Yaskawa INFORM job: X2_38-47,64(2)(90,0)_HARDOX.JBI

/JOB
//NAME X2_38-47,64(2)(90,0)_HARDOX
//POS
///NPOS 517,517,517,31,0,0
///TOOL 0
///POSTYPE PULSE
///PULSE
C00000=-10776,-116726,-133110,1428,79202,268
C00001=-117551,-99167,-129064,14869,107235,27560
C00002=-118060,-97833,-124544,14759,105287,27149
C00003=-118255,-97731,-122391,14687,104086,26936
C00004=-118255,-99005,-121658,14606,103015,26804
C00005=-118252,-98719,-121832,14623,103261,26835
C00006=-118753,-92238,-119382,14829,105109,26899
C00007=-118252,-98719,-121832,14623,103261,26835
C00008=-117548,-101379,-128390,14732,105732,27372
C00009=-119930,-99721,-129265,15188,107465,26816
C00010=-120369,-98285,-124713,15062,105542,26424
C00011=-120537,-98252,-122491,14975,104264,26206
C00012=-120537,-99415,-121812,14899,103281,26083
C00013=-120552,-99088,-121997,14922,103557,26112
C00014=-120983,-92542,-119530,15124,105413,26206
C00015=-120552,-99088,-121997,14922,103557,26112
C00016=-119945,-101871,-128593,15052,105999,26622
C00017=-126449,-117484,-130445,19479,74849,30062
C00018=-126433,-122162,-123583,20167,68593,29001
C00019=-126700,-111661,-117040,20113,69946,29141
C00020=-126798,-108107,-114012,20160,69935,29102
C00021=-126799,-108400,-113008,20254,69212,28975
C00022=-126718,-108336,-113627,20168,69582,29070
C00023=-124486,-105728,-112699,19107,69790,29924
C00024=-126718,-108336,-113627,20168,69582,29070
C00025=-121607,-132044,-121280,18982,61321,29585
C00026=-106120,-105771,-112642,10491,66484,36125
C00027=-107709,-101450,-111061,11179,67916,35692
C00028=-106120,-105771,-112642,10491,66484,36125
C00029=-113778,-131562,-126460,14735,63009,32904
C00030=-125989,-135705,-128836,15868,81833,-19678
C00031=-122637,-125595,-122855,15098,82666,-18409
C00032=-121382,-121958,-120533,14807,82865,-17952
C00033=-121382,-122071,-118910,14836,81841,-18076
C00034=-121382,-121958,-120533,14807,82865,-17952
C00035=-106979,-143901,-125029,2861,68009,-11090
C00036=-108002,-136905,-123073,3147,70435,-11396
C00037=-106979,-143901,-125029,2861,68009,-11090
C00038=-130918,-93362,-108301,23503,98063,-21430
C00039=-128613,-93045,-108174,23197,97523,-20724
C00040=-130918,-93362,-108301,23503,98063,-21430
C00041=-136165,-97259,-113946,24281,100844,-22722
C00042=-136175,-89641,-119549,25205,107565,-21267
C00043=-114744,-130738,-127344,-18726,86415,24127
C00044=-118651,-123075,-122041,-18017,86194,22796
C00045=-120132,-120263,-119410,-17742,85711,22351
C00046=-120132,-120365,-118339,-17753,85031,22450
C00047=-120131,-120316,-118616,-17749,85218,22423
C00048=-120610,-114014,-116540,-17635,86988,22001
C00049=-120131,-120316,-118616,-17749,85218,22423
C00050=-120535,-116966,-117470,-17658,86102,22155
C00051=-123144,-118008,-117813,-17156,85246,21372
C00052=-120535,-116966,-117470,-17658,86102,22155
C00053=-115268,-126863,-124750,-18631,86672,23904
C00054=-115290,-123417,-132013,-18678,92595,22992
C00055=-123593,-125758,-130163,6995,115060,-67946
C00056=-111289,-112434,-124190,9231,117016,-63234
C00057=-105837,-112853,-120878,9823,114178,-61462
C00058=-105837,-113368,-119803,9744,113264,-61541
C00059=-105837,-112984,-120626,9804,113958,-61481
C00060=-104314,-115180,-121361,9954,113110,-60999
C00061=-105837,-112984,-120626,9804,113958,-61481
C00062=-140180,-156270,-135194,3647,103600,-74458
C00063=-143876,-158808,-133483,2421,103143,-75779
C00064=-143876,-157752,-132173,2418,102880,-75785
C00065=-143876,-158999,-133717,2421,103190,-75779
C00066=-142833,-166242,-135523,2599,100548,-75469
C00067=-143876,-158999,-133717,2421,103190,-75779
C00068=-138517,-137739,-134524,3768,114393,-73549
C00069=-143641,-117492,-131018,10110,103710,-40081
C00070=-127017,-112123,-129453,9078,98380,-24722
C00071=-128303,-122732,-125182,9622,82824,-11347
C00072=-126354,-112603,-118881,9097,83916,-10616
C00073=-125631,-108986,-116438,8904,84188,-10357
C00074=-125631,-109537,-114964,8919,83013,-10441
C00075=-125631,-108986,-116438,8904,84188,-10357
C00076=-110037,-120252,-118594,-5441,76700,-4050
C00077=-111650,-115152,-116920,-4919,78183,-4659
C00078=-110037,-120252,-118594,-5441,76700,-4050
C00079=-125797,-107165,-114352,8951,83863,-10435
C00080=-123589,-104463,-113383,8361,84418,-9668
C00081=-125797,-107165,-114352,8951,83863,-10435
C00082=-128447,-120300,-122969,9661,82730,-11402
C00083=-128462,-115265,-129707,9620,89375,-10895
C00084=-116938,-126430,-125851,-12631,81878,14685
C00085=-119474,-116309,-119688,-11957,82879,13726
C00086=-120416,-112800,-116898,-11714,82830,13413
C00087=-120416,-113088,-115771,-11732,82005,13491
C00088=-121130,-109897,-115487,-11517,83341,13125
C00089=-121652,-107697,-114715,-11371,83913,12898
C00090=-120385,-110630,-116263,-11708,83544,13356
C00091=-116898,-126708,-125088,-12658,81285,14759
C00092=-116961,-121523,-133241,-12544,88781,13978
C00093=-110477,-156196,-127656,-40514,54336,55405
C00094=-116757,-147091,-123275,-37008,53079,52657
C00095=-119129,-143495,-121504,-35581,52690,51595
C00096=-122199,-143523,-121511,-34086,51426,50520
C00097=-119129,-143495,-121504,-35581,52690,51595
C00098=-121389,-143526,-121523,-34489,51757,50806
C00099=-121378,-138155,-118828,-34021,52680,50458
C00100=-121389,-143526,-121523,-34489,51757,50806
C00101=-121337,-120057,-120260,-30579,61379,47564
C00102=-120272,-114318,-116759,-30898,62447,47698
C00103=-120254,-119054,-117181,-31500,60580,48280
C00104=-120272,-114318,-116759,-30898,62447,47698
C00105=-110477,-159292,-131347,-40206,54861,55162
C00106=-115322,-144881,-127675,-10917,26238,44128
C00107=-131784,-127965,-127002,28991,89678,26741
C00108=-120831,-123140,-121731,27130,85392,29797
C00109=-120549,-120601,-118843,27089,84879,29783
C00110=-120549,-120670,-117777,27109,84260,29640
C00111=-120517,-120686,-117908,27101,84315,29665
C00112=-120983,-114470,-115866,27142,86197,29928
C00113=-120517,-120686,-117908,27101,84315,29665
C00114=-121539,-130455,-126219,27290,84728,29379
C00115=-123491,-138727,-133578,17593,86073,29901
C00116=-123873,-130565,-127363,17655,86508,29830
C00117=-124019,-127789,-124130,17687,86001,29706
C00118=-124019,-127817,-123341,17694,85524,29637
C00119=-124041,-127842,-123499,17696,85609,29642
C00120=-124402,-120732,-121277,17740,87868,29843
C00121=-124041,-127842,-123499,17696,85609,29642
C00122=-123895,-130695,-125894,17671,85585,29689
C00123=-123514,-138829,-132098,17610,85158,29761
C00124=-131669,-108309,-130646,31875,113573,61343
C00125=-139138,-132176,-121475,37127,109735,76690
C00126=-136347,-141301,-121131,36509,104575,76083
C00127=-135137,-144527,-120818,36387,102556,75910
C00128=-135139,-143303,-118803,36292,102059,75739
C00129=-135137,-144527,-120818,36387,102556,75910
C00130=-123222,-117207,-112602,33876,112841,80142
C00131=-123302,-123100,-114500,33386,111310,79603
C00132=-123222,-117207,-112602,33876,112841,80142
C00133=-149473,-167599,-122340,40123,93659,70303
C00134=-145955,-169881,-122827,40768,91382,70949
C00135=-149473,-167599,-122340,40123,93659,70303
C00136=-154660,-158984,-124630,39692,100555,70658
C00137=-145602,-129354,-130944,11561,117970,66438
C00138=-141571,-135796,-129141,-17923,112920,58745
C00139=-145358,-145317,-128855,-18021,107261,58200
C00140=-146973,-148537,-128532,-18134,105137,57926
C00141=-146977,-147425,-126561,-18072,104525,58019
C00142=-146951,-147398,-126788,-18082,104677,58005
C00143=-148016,-155121,-128806,-18044,101844,58047
C00144=-146951,-147398,-126788,-18082,104677,58005
C00145=-147811,-154474,-129578,-18071,102659,57998
C00146=-150760,-151393,-128781,-18698,103033,56852
C00147=-147811,-154474,-129578,-18071,102659,57998
C00148=-142197,-142429,-130522,-17697,110344,58914
C00149=-120703,-123129,-132845,19094,121060,67264
C00150=-120658,-146832,-128060,18624,118943,66884
C00151=-120634,-158899,-128202,17585,113113,65913
C00152=-120623,-163194,-128036,17271,110903,65572
C00153=-120623,-161024,-125795,17237,110651,65534
C00154=-120562,-161261,-126266,17282,110799,65580
C00155=-120543,-169070,-128088,16945,108025,65171
C00156=-120562,-161261,-126266,17282,110799,65580
C00157=-120603,-145779,-126506,18564,118536,66834
C00158=-125859,-133715,-124767,32608,106843,81797
C00159=-122845,-142953,-124347,32149,101432,81430
C00160=-121547,-146160,-123992,32074,99345,81353
C00161=-121546,-144979,-121994,32008,98813,81200
C00162=-109812,-115651,-114700,28773,111647,86169
C00163=-109420,-121743,-116686,28433,109829,85843
C00164=-109812,-115651,-114700,28773,111647,86169
C00165=-136113,-171916,-125823,37236,88758,74782
C00166=-132431,-173177,-126093,37775,86796,75630
C00167=-136113,-171916,-125823,37236,88758,74782
C00168=-141699,-164023,-128432,36630,95711,74814
C00169=-125872,-133752,-131219,33440,110189,40846
C00170=-133109,-126295,-132836,15576,121717,-49477
C00171=-134095,-144484,-127159,11413,120192,-39245
C00172=-134095,-142728,-123587,11251,118920,-39381
C00173=-134108,-141028,-121891,11256,119008,-39376
C00174=-115660,-122947,-115610,-13186,126131,-57848
C00175=-119844,-134491,-118750,-17115,121000,-60623
C00176=-133528,-137451,-116046,-34139,108998,-80448
C00177=-134077,-138654,-116284,-35996,107959,-82962
C00178=-134074,-140235,-119255,-36225,108790,-83252
C00179=-128746,-104991,-133081,-28169,117444,-49732
C00180=-123335,-90933,-122081,-14660,102496,-9308
C00181=-120623,-92535,-112214,-7385,88125,11837
C00182=-120622,-94347,-109953,-7392,85821,11972
C00183=-121706,-96320,-109727,-7087,84579,11689
C00184=-119347,-92925,-108176,-7759,85570,12397
C00185=-120623,-94767,-108750,-7400,84873,12029
C00186=-120184,-98406,-104184,11463,70199,-7234
C00187=-120621,-97250,-102226,16251,67423,-11647
C00188=-120622,-96877,-104163,16104,68755,-11460
C00189=-120643,-108357,-118989,16415,66098,-11840
C00190=-67024,-106779,-124945,-13769,92672,20129
C00191=-67015,-109280,-122780,-13735,90127,20415
C00192=-68524,-114997,-123393,-13374,87393,20218
C00193=-67240,-109374,-121326,-13663,89172,20449
C00194=-67101,-109000,-122679,-13716,90193,20379
C00195=-67110,-106486,-124839,-13750,92741,20094
C00196=-120616,-103713,-129855,-8435,78518,79847
C00197=-120615,-108904,-127553,-8566,74477,80127
C00198=-120827,-110646,-126375,-8530,72852,80171
C00199=-120813,-110572,-126430,-8535,72927,80169
C00200=-120709,-110247,-126307,-8582,73030,80199
C00201=-120779,-110557,-126444,-8550,72945,80181
C00202=-120615,-108909,-127550,-8566,74473,80128
C00203=-118661,-125998,-116417,-35444,53464,49551
C00204=-120918,-122974,-114552,-34038,52889,48644
C00205=-120869,-128815,-114683,-35350,50480,49611
C00206=-120575,-146473,-114035,-40240,44023,53993
C00207=-120599,-119966,-113452,-30276,65744,57931
C00208=-118319,-121507,-115012,-31110,66714,58605
C00209=-113281,-124998,-118777,-32819,69049,60013
C00210=-113467,-117261,-128448,-33027,70743,59318
C00211=-117537,-116112,-134646,-12805,84442,25722
C00212=-120610,-126431,-125414,1040,80197,3464
C00213=-120610,-126707,-122448,1046,78230,3447
C00214=-122238,-127010,-121321,1494,77406,2886
C00215=-120610,-126687,-121221,1049,77486,3441
C00216=-120610,-126294,-121087,1045,77585,3442
C00217=-120610,-126285,-120333,4549,75913,-5215
C00218=-120610,-126340,-121533,4537,76621,-5189
C00219=-125895,-134934,-128716,6057,76967,-6982
C00220=-120648,-124280,-131590,4464,45149,-4941
C00221=-120660,-101129,-132257,5341,102721,-45112
C00222=-120607,-133883,-126281,5735,119700,-79532
C00223=-120606,-133398,-123219,5634,118073,-79618
C00224=-121083,-132569,-121808,5443,117663,-79827
C00225=-120607,-132621,-121847,5608,117630,-79641
C00226=-120606,-132785,-121826,5603,117534,-79644
C00227=-120606,-132451,-120233,13920,116954,-67409
C00228=-120606,-132780,-121444,14001,117514,-67337
C00229=-120606,-133413,-124386,14219,118956,-67146
C00230=-118302,-128282,-130929,25956,92288,-30440
C00231=-120609,-125694,-119256,16594,71477,-14811
C00232=-120609,-125321,-116628,16727,70109,-15005
C00233=-120267,-125069,-115718,16650,69625,-14949
C00234=-120609,-125952,-120025,-8845,76809,6022
C00235=-120609,-125682,-119997,-8842,76927,6012
C00236=-120946,-125172,-117915,-18180,76717,18969
C00237=-120609,-125456,-118894,-18238,77226,19012
C00238=-120610,-125544,-121647,-18141,78796,18775
C00239=-120644,-111765,-129409,-18832,94472,5338
C00240=-120647,-108820,-131188,-26213,120818,-60808
C00241=-120603,-141811,-125437,-24145,112419,-84195
C00242=-120603,-140407,-122244,-23914,111279,-83943
C00243=-120716,-139436,-120851,-23880,110920,-83910
C00244=-120603,-141515,-124307,-1,115345,-75490
C00245=-120603,-141196,-124279,-1,115492,-75490
C00246=-120750,-138616,-117883,30210,107343,-65244
C00247=-120602,-139074,-119094,30337,107734,-65073
C00248=-120603,-140473,-121905,30531,108612,-64825
C00249=-123038,-137969,-128708,31970,112888,-64779
C00250=-147472,-118060,-121113,40576,103304,-81843
C00251=-147472,-118630,-118217,40218,101703,-82475
C00252=-147472,-118727,-117017,40094,101093,-82713
C00253=-147408,-115266,-125424,616,120610,-87255
C00254=-147440,-115512,-125518,608,120541,-87267
C00255=-147454,-115617,-125558,7144,119076,-75809
C00256=-147463,-115686,-125590,12209,115534,-64774
C00257=-147467,-115708,-125608,15036,110623,-54333
C00258=-147465,-115687,-125611,15580,106535,-46817
C00259=-147461,-115654,-125607,15271,104034,-42312
C00260=-147458,-115622,-125603,14500,101619,-37854
C00261=-147455,-115603,-125598,14501,101625,-37852
C00262=-147455,-114670,-126645,14574,102714,-37720
C00263=-147454,-112308,-128585,14752,105047,-37432
C00264=-120607,-127649,-132770,-5702,79300,5510
C00265=-120610,-123519,-126906,-5727,77820,5577
C00266=-120610,-124347,-124400,-5769,75861,5668
C00267=-121328,-123636,-123053,-5535,75349,5445
C00268=-120611,-123827,-123148,-12249,77590,12361
C00269=-120610,-124176,-124804,-8835,80309,9900
C00270=-120610,-124421,-124355,885,77124,6939
C00271=-120609,-123606,-124090,-1533,77411,9469
C00272=-116475,-118028,-122311,-2829,79291,10818
C00273=-112174,-113451,-120859,-4161,80928,12195
C00274=-109550,-110906,-119998,-4966,81848,13023
C00275=-120610,-123835,-125318,-1528,78049,9462
C00276=-120610,-122990,-127374,-1521,79748,9441
C00277=2000,-133752,-131219,0,47993,0
C00278=-63459,-114373,-79771,19626,40886,37257
C00279=-120535,67520,37147,4212,69072,67068
C00280=-120830,69446,43417,4422,66227,66858
C00281=-120946,70374,46117,4513,65052,66770
C00282=-120946,70561,47998,4551,63994,66728
C00283=-120946,70374,46117,4513,65052,66770
C00284=-120262,65088,41656,4214,65044,67021
C00285=-120723,68225,45319,4437,64429,66828
C00286=-120262,65088,41656,4214,65044,67021
C00287=-120141,64198,39022,4125,66199,67107
C00288=-119837,62342,32876,3917,69006,67311
C00289=-133022,42545,9302,483,69993,74705
C00290=-133254,43745,14595,601,67354,74612
C00291=-133346,44332,16823,649,66285,74574
C00292=-133347,44228,18372,654,65278,74568
C00293=-133346,44332,16823,649,66285,74574
C00294=-132762,39917,13904,373,65809,74781
C00295=-133123,42775,16905,546,65433,74650
C00296=-132762,39917,13904,373,65809,74781
C00297=-132666,39314,11672,325,66873,74819
C00298=-132425,38068,6360,208,69500,74909
C00299=-155117,5532,-38436,2147,90846,73739
C00300=-181330,90113,53999,1695,94832,75162
C00301=-181479,87228,54387,1703,93114,75089
C00302=-181540,86155,54651,1706,92402,75059
C00303=-181542,86152,56307,1705,91382,75044
C00304=-181540,86155,54651,1706,92402,75059
C00305=-180656,94851,65604,1626,90111,75325
C00306=-181131,94253,66558,1666,89229,75153
C00307=-181349,89885,61022,1686,90394,75096
C00308=-181131,94253,66558,1666,89229,75153
C00309=-181073,95243,66217,1662,89945,75182
C00310=-180930,97948,65680,1651,91663,75253
C00311=-185436,101694,69046,-5553,88631,72150
C00312=-185900,99624,70331,-5496,86754,72076
C00313=-186037,103761,77290,-5473,84596,72123
C00314=-186037,104195,79283,-5480,83598,72167
C00315=-186037,104106,78898,-5479,83788,72160
C00316=-185971,101194,75107,-5481,84626,72147
C00317=-185574,103041,75706,-5528,85231,72255
C00318=-185712,103515,76702,-5528,84853,72223
C00319=-185252,105372,75160,-5578,86780,72294
C00320=-160848,14099,-19058,-268,71131,81958
C00321=-166181,22945,-3449,-1246,81387,-4932
C00322=-165629,27427,7007,-1415,77267,-4702
C00323=-165325,28785,10065,-1509,76088,-4584
C00324=-165325,28859,11250,-1513,75397,-4577
C00325=-165325,28785,10065,-1509,76088,-4584
C00326=-165316,31705,12964,-1515,75805,-4576
C00327=-165325,28785,10065,-1509,76088,-4584
C00328=-158615,35277,16566,-12881,79402,10247
C00329=-158695,35491,17753,-12887,78784,10285
C00330=-159268,36430,18712,-12762,78589,10105
C00331=-158695,35389,16453,-12860,79513,10210
C00332=-158695,35595,7262,-12723,85139,9628
C00333=-159201,23460,163,-1108,64126,82575
C00334=-159224,25290,5934,-1122,61515,82592
C00335=-159102,29806,11901,-1198,60164,82651
C00336=-159102,29893,13040,-1208,59512,82655
C00337=-159102,29869,12753,-1208,59677,82655
C00338=-159322,25425,8401,-1088,60068,82565
C00339=-159448,23983,7363,-1023,59965,82516
C00340=-159276,26818,10107,-1116,59735,82583
C00341=-159294,26208,9511,-1106,59788,82576
C00342=-159294,26230,9792,-1106,59626,82576
C00343=-159101,23920,6361,-1196,60552,82648
C00344=-159295,23244,6238,-1098,60277,82577
C00345=-159295,23301,7050,-1101,59807,82580
C00346=-159299,25281,8955,-1100,59652,82580
C00347=-159295,23278,6733,-1101,59990,82580
C00348=-159427,17860,-3265,-1001,63356,82499
C00349=-180998,44453,11386,9428,69103,75000
C00350=-180806,46143,18147,9552,65832,74803
C00351=-180618,49143,21508,9515,65295,74827
C00352=-180618,49076,22901,9581,64417,74754
C00353=-180618,49087,22593,9566,64610,74771
C00354=-181106,45329,18547,9757,65218,74643
C00355=-181106,45312,18870,9772,65014,74625
C00356=-180958,47165,20854,9721,64729,74655
C00357=-180909,46562,20206,9690,64811,74680
C00358=-180909,46552,20476,9701,64642,74667
C00359=-180909,46563,20203,9689,64813,74682
C00360=-181219,43931,17395,9810,65220,74603
C00361=-181219,43906,17870,9834,64920,74577
C00362=-181012,45777,19861,9753,64635,74629
C00363=-181381,44679,17515,9863,65546,74571
C00364=-181427,38720,7071,9647,68865,74830
C00365=-194866,69356,39319,16134,66946,69768
C00366=-193573,77344,52867,16088,62620,69643
C00367=-194003,72673,48449,16239,63021,69537
C00368=-194003,72898,50393,16388,61984,69385
C00369=-194003,72870,50176,16371,62099,69402
C00370=-193870,75079,52821,16382,61600,69380
C00371=-193864,70129,44405,16015,64135,69754
C00372=-195158,66932,37846,16301,66678,69622
C00373=-181592,-32488,-72920,9217,81357,75741
C00374=-150216,-104680,-71296,-7403,42753,75254
C00375=-146927,-106152,-71782,-9593,42642,76873
C00376=-147684,-69879,-51768,-13743,41767,65179
C00377=-160676,17315,-11357,-3352,97353,79993
C00378=-160891,14623,-4117,-3294,91515,80076
C00379=-160979,13901,-3035,-3283,90476,80074
C00380=-160979,13973,-1608,-3282,89636,80096
C00381=-160979,13952,-1963,-3282,89844,80091
C00382=-161075,20354,3961,-3273,89483,80067
C00383=-161075,20386,4410,-3273,89224,80073
C00384=-161133,18273,2432,-3268,89353,80049
C00385=-161218,18655,2789,-3260,89326,80020
C00386=-161218,18671,3009,-3260,89200,80024
C00387=-161218,18657,2809,-3260,89316,80021
C00388=-161242,21197,5196,-3258,89153,80017
C00389=-161242,21225,5559,-3258,88944,80022
C00390=-161222,19566,3996,-3259,89054,80025
C00391=-161093,20062,3160,-3271,89826,80048
C00392=-160610,22295,943,-3323,92353,80148
C00393=-159769,-26352,-42847,7626,75430,42908
C00394=-160661,-23608,-37245,8003,73495,42476
C00395=-161092,-17751,-31188,8180,72827,42281
C00396=-161092,-17734,-30227,8206,72247,42243
C00397=-161092,-17740,-30493,8199,72405,42254
C00398=-161118,-21273,-33081,8218,72187,42230
C00399=-161118,-21265,-32749,8226,71987,42217
C00400=-161116,-19976,-31814,8223,72071,42223
C00401=-161133,-20273,-32030,8231,72055,42216
C00402=-161133,-20265,-31761,8239,71896,42206
C00403=-161133,-20272,-31998,8233,72037,42215
C00404=-161051,-23031,-33989,8213,71838,42230
C00405=-161051,-23018,-33649,8222,71636,42217
C00406=-160924,-21492,-32553,8173,71734,42269
C00407=-161101,-22161,-33921,8213,72245,42241
C00408=-159612,-30937,-44211,7622,73912,42867
C00409=-147684,-69879,-51768,-13743,41767,65179
C00410=-146927,-106152,-71782,-9593,42642,76873
C00411=-150216,-104680,-71296,-7403,42753,75254
C00412=-181592,-37651,-66165,9425,74633,75233
C00413=-161871,17303,-4712,10555,76262,79929
C00414=-161452,17546,-388,10536,73713,79854
C00415=-164352,5532,-4911,18132,62198,77732
C00416=-162815,5376,-4950,17454,61813,78279
C00417=-160145,17568,-217,10119,73455,80292
C00418=-160561,17295,-4569,10141,76006,80359
C00419=-160561,17295,-4569,10141,77854,24225
C00420=-154925,3428,-11232,-4624,70900,30462
C00421=-155821,5540,-7163,-4340,69436,30196
C00422=-157012,4626,-7218,-1589,68724,27505
C00423=-155631,5235,-4373,-2115,67316,28026
C00424=-155501,1121,-9941,-2144,68631,28049
C00425=-164062,1653,-9261,9806,70969,1365
C00426=-163111,13453,569,7852,75819,2004
C00427=-169111,38169,24298,20475,87264,-21600
C00428=-171145,34811,19304,20623,89038,-22029
C00429=-170232,24106,-2783,18479,91787,-14288
C00430=-160304,11530,-9767,5228,51358,81447
C00431=-160077,14832,-4280,5183,49670,81455
C00432=-160516,13652,-395,8281,43180,80940
C00433=-159075,15987,128,5765,45857,81735
C00434=-164330,15419,2317,23639,44338,76758
C00435=-163385,18960,-1174,18743,50959,78553
C00436=-165374,13239,-6613,20923,51920,77727
C00437=-161014,13295,-8090,-6406,49355,82824
C00438=-161267,16828,-2191,-6383,47532,82835
C00439=-161514,15522,988,-4927,41294,83331
C00440=-163506,13156,714,-1971,37859,82561
C00441=-158654,13018,2647,-21114,36743,89145
C00442=-156013,15323,-3292,-22041,49335,86873
C00443=-155829,15379,-4520,-22688,50226,86879
C00444=-196408,57492,27109,18880,55161,68375
C00445=-196116,61126,34099,19257,52786,68047
C00446=-196624,61095,37640,23439,48900,67243
C00447=-198066,64493,41377,24271,49005,66556
C00448=-198035,64746,39034,20821,52142,67068
C00449=-198350,60950,31019,20265,55020,67530
C00450=-186747,89870,54733,-990,89142,72486
C00451=-186403,90906,60090,-1045,86383,72625
C00452=-181702,120366,100649,-11275,85103,73801
C00453=-183712,129983,113842,-11249,81700,73410
C00454=-188822,91256,60525,-666,86269,71815
C00455=-188503,92942,58606,-716,88318,71911
C00456=-158356,2052,-43381,6178,92005,68050
C00457=-121453,57439,26725,6551,67570,68970
C00458=-121610,59341,32873,6761,64794,68755
C00459=-121469,44825,24088,7614,53384,68067
C00460=-119406,47984,28011,6377,51946,68833
C00461=-119643,63560,37702,5874,63844,69428
C00462=-119474,61501,31338,5667,66676,69631
C00463=-119468,73784,45718,-1688,68030,70001
C00464=-119896,75838,52185,-1543,65099,69887
C00465=-119734,60370,40471,-1882,55599,70088
C00466=-120784,60524,39839,-1249,57371,69644
C00467=-121139,72676,48393,-1011,65788,69424
C00468=-120714,70771,42130,-1166,68668,69550
C00469=-130022,48445,16791,-5635,70294,75741
C00470=-130464,49596,22041,-5533,67637,75710
C00471=-130594,37241,15185,-4965,57340,76243
C00472=-134757,36577,12787,-2863,61070,74469
C00473=-134997,44020,16033,-3483,68218,74080
C00474=-134574,42926,10871,-3614,70846,74149
C00475=-144116,-100954,-108623,608,70277,70877
C00476=-125234,-105855,-90971,-8573,57832,78294
C00477=-134723,-30987,-43000,-16193,82094,-73445
C00478=-147286,-18641,-32771,2207,85620,-76456
C00479=-145987,-10544,-25760,-132,91452,-76157
C00480=-145688,-12541,-27327,264,90178,-76022
C00481=-146939,-19097,-33105,2145,85581,-76340
C00482=-147575,-22440,-39612,2256,87884,-76511
C00483=-160185,17986,-3976,-6942,87400,-80225
C00484=-159579,20779,2718,-7055,84786,-79877
C00485=-159753,19362,2506,-7031,84177,-79901
C00486=-161023,19371,2516,-6819,84070,-80326
C00487=-160409,20517,1737,-6914,85180,-80178
C00488=-160981,17969,-3994,-6807,87335,-80488
C00489=-162074,-26616,-42506,-1763,64705,-79693
C00490=-162070,-24854,-37261,-1799,62384,-79656
C00491=-162357,-21732,-33702,-1661,61789,-79757
C00492=-160326,-21798,-33765,-2703,61848,-78996
C00493=-159769,-24818,-37192,-4027,62449,-78761
C00494=-159682,-26579,-42435,-3993,64769,-78811
C00495=-159749,-26590,-42466,-830,64636,-81339
C00496=-159773,-24828,-37221,-834,62313,-81331
C00497=-159460,-21788,-33850,-1000,61804,-81209
C00498=-160671,-21843,-33924,-379,61812,-81664
C00499=-162116,-24842,-37231,1419,62318,-82243
C00500=-162183,-26603,-42475,1425,64641,-82238
C00501=-125234,-105855,-90971,-8573,57832,78294
C00502=-144116,-100954,-108623,608,70277,70877
C00503=-180054,17730,-13564,7282,57092,75133
C00504=-184405,44193,24876,11651,47654,72434
C00505=-186318,42466,29434,20119,40097,70434
C00506=-189623,46674,33918,23221,40411,68696
C00507=-188153,48497,30967,14785,46766,70568
C00508=-188342,44346,22853,14289,49572,70918
C00509=-179348,87345,51596,-2140,89915,74922
C00510=-179393,86533,54635,-2132,87627,74946
C00511=-176610,100170,73501,-7799,88743,75470
C00512=-180322,105518,80466,-7431,86799,74328
C00513=-183307,90153,59154,-1526,86619,73655
C00514=-183010,91971,57396,-1572,88641,73729
C00515=-153116,42547,-17943,-6513,110885,24646
C00516=-10907,-117335,-90652,-18762,63715,-59495
BC00000=165820,667836,1075229
BC00001=398174,1010261,1075175
BC00002=398174,1010261,1075175
BC00003=398174,1010261,1075175
BC00004=398174,1010261,1075175
BC00005=398174,1010261,1075175
BC00006=398174,1010261,1075175
BC00007=398174,1010261,1075175
BC00008=398174,1010261,1075175
BC00009=355157,1002325,1075175
BC00010=355157,1002325,1075175
BC00011=355157,1002325,1075175
BC00012=355157,1002325,1075175
BC00013=355157,1002325,1075175
BC00014=355157,1002325,1075175
BC00015=355157,1002325,1075175
BC00016=355157,1002325,1075175
BC00017=253987,909376,1075175
BC00018=253987,909376,1075175
BC00019=253987,909376,1075175
BC00020=253987,909376,1075175
BC00021=253987,909376,1075175
BC00022=253987,909376,1075175
BC00023=253987,909376,1075175
BC00024=253987,909376,1075175
BC00025=253987,909376,1075175
BC00026=253987,909376,1075175
BC00027=253987,909376,1075175
BC00028=253987,909376,1075175
BC00029=253987,909376,1075175
BC00030=147037,948855,1075175
BC00031=147037,948855,1075175
BC00032=147037,948855,1075175
BC00033=147037,948855,1075175
BC00034=147037,948855,1075175
BC00035=147037,948855,1075175
BC00036=147037,948855,1075175
BC00037=147037,948855,1075175
BC00038=147037,948855,1075175
BC00039=147037,948855,1075175
BC00040=147037,948855,1075175
BC00041=147037,948855,1075175
BC00042=147037,948855,1075175
BC00043=175618,946621,1075175
BC00044=175618,946621,1075175
BC00045=175618,946621,1075175
BC00046=175618,946621,1075175
BC00047=175618,946621,1075175
BC00048=175618,946621,1075175
BC00049=175618,946621,1075175
BC00050=175618,946621,1075175
BC00051=175618,946621,1075175
BC00052=175618,946621,1075175
BC00053=175618,946621,1075175
BC00054=175618,946621,1075175
BC00055=144312,974949,1075175
BC00056=144312,974949,1075175
BC00057=144312,974949,1075175
BC00058=144312,974949,1075175
BC00059=144312,974949,1075175
BC00060=144312,974949,1075175
BC00061=144312,974949,1075175
BC00062=144312,974949,1075175
BC00063=144312,974949,1075175
BC00064=144312,974949,1075175
BC00065=144312,974949,1075175
BC00066=144312,974949,1075175
BC00067=144312,974949,1075175
BC00068=144312,974949,1075175
BC00069=159928,928652,1075175
BC00070=164440,875523,1075175
BC00071=171034,862645,1075175
BC00072=171034,862645,1075175
BC00073=171034,862645,1075175
BC00074=171034,862645,1075175
BC00075=171034,862645,1075175
BC00076=171034,862645,1075175
BC00077=171034,862645,1075175
BC00078=171034,862645,1075175
BC00079=171034,862645,1075175
BC00080=171034,862645,1075175
BC00081=171034,862645,1075175
BC00082=171034,862645,1075175
BC00083=171034,862645,1075175
BC00084=164738,841983,1075175
BC00085=164738,841983,1075175
BC00086=164738,841983,1075175
BC00087=164738,841983,1075175
BC00088=164738,841983,1075175
BC00089=164738,841983,1075175
BC00090=164738,841983,1075175
BC00091=164738,841983,1075175
BC00092=164738,841983,1075175
BC00093=143339,934688,1075175
BC00094=143339,934688,1075175
BC00095=143339,934688,1075175
BC00096=143339,934688,1075175
BC00097=143339,934688,1075175
BC00098=143339,934688,1075175
BC00099=143339,934688,1075175
BC00100=143339,934688,1075175
BC00101=143339,934688,1075175
BC00102=143339,934688,1075175
BC00103=143339,934688,1075175
BC00104=143339,934688,1075175
BC00105=143339,934688,1075175
BC00106=95192,864025,1075175
BC00107=33067,951094,1075175
BC00108=33067,951094,1075175
BC00109=33067,951094,1075175
BC00110=33067,951094,1075175
BC00111=33067,951094,1075175
BC00112=33067,951094,1075175
BC00113=33067,951094,1075175
BC00114=33067,951094,1075175
BC00115=15,945322,1075175
BC00116=15,945322,1075175
BC00117=15,945322,1075175
BC00118=15,945322,1075175
BC00119=15,945322,1075175
BC00120=15,945322,1075175
BC00121=15,945322,1075175
BC00122=15,945322,1075175
BC00123=15,945322,1075175
BC00124=16460,857819,1075175
BC00125=28300,807028,1075175
BC00126=28300,807028,1075175
BC00127=28300,807028,1075175
BC00128=28300,807028,1075175
BC00129=28300,807028,1075175
BC00130=28300,807028,1075175
BC00131=28300,807028,1075175
BC00132=28300,807028,1075175
BC00133=28300,807028,1075175
BC00134=28300,807028,1075175
BC00135=28300,807028,1075175
BC00136=28300,807028,1075175
BC00137=49949,826856,1075175
BC00138=70323,828866,1075175
BC00139=70323,828866,1075175
BC00140=70323,828866,1075175
BC00141=70323,828866,1075175
BC00142=70323,828866,1075175
BC00143=70323,828866,1075175
BC00144=70323,828866,1075175
BC00145=70323,828866,1075175
BC00146=70323,828866,1075175
BC00147=70323,828866,1075175
BC00148=70323,828866,1075175
BC00149=113400,816475,1075175
BC00150=113400,846295,1075175
BC00151=113400,846295,1075175
BC00152=113400,846295,1075175
BC00153=113400,846295,1075175
BC00154=113400,846295,1075175
BC00155=113400,846295,1075175
BC00156=113400,846295,1075175
BC00157=113400,846295,1075175
BC00158=126179,809480,1075175
BC00159=126179,809480,1075175
BC00160=126179,809480,1075175
BC00161=126179,809480,1075175
BC00162=126179,809480,1075175
BC00163=126179,809480,1075175
BC00164=126179,809480,1075175
BC00165=126179,809480,1075175
BC00166=126179,809480,1075175
BC00167=126179,809480,1075175
BC00168=126179,809480,1075175
BC00169=126179,809480,1075175
BC00170=153260,992688,1075175
BC00171=154894,1008954,1075175
BC00172=159567,1006428,1075175
BC00173=161040,1005633,1075171
BC00174=188180,1004944,1075172
BC00175=159398,988729,1075171
BC00176=196171,985949,1075168
BC00177=201136,987895,1075175
BC00178=203670,993516,1075175
BC00179=184106,924906,1075175
BC00180=164145,855826,1075175
BC00181=154136,821185,1075175
BC00182=151914,826190,1075175
BC00183=151025,828192,1075175
BC00184=151025,828192,1075175
BC00185=197574,854331,1075175
BC00186=160004,840173,1075175
BC00187=151157,834851,1075175
BC00188=148293,828805,1075175
BC00189=148293,828805,1075175
BC00190=312275,994515,1075175
BC00191=311979,999858,1075175
BC00192=311860,1001996,1075175
BC00193=362733,1010828,1075164
BC00194=362852,1008691,1075175
BC00195=363148,1003347,1075175
BC00196=102795,934804,1075175
BC00197=101452,936777,1075175
BC00198=100915,937567,1075175
BC00199=100906,939899,1075175
BC00200=100898,942175,1075175
BC00201=100889,944507,1075175
BC00202=101426,943718,1075175
BC00203=141515,928256,1075175
BC00204=141515,928256,1075175
BC00205=141515,928256,1075175
BC00206=141515,928257,1075172
BC00207=141515,928256,1075175
BC00208=141515,928256,1075175
BC00209=141515,928256,1075175
BC00210=141515,916104,1075175
BC00211=68127,920356,1075175
BC00212=16830,923328,1075175
BC00213=16562,928525,1075175
BC00214=16455,930603,1075175
BC00215=16455,930603,1075175
BC00216=71893,940191,1075175
BC00217=67464,939156,1075175
BC00218=67022,937046,1075175
BC00219=65915,931769,1075175
BC00220=65915,901978,1075175
BC00221=98323,852136,1075175
BC00222=125079,831224,1075175
BC00223=125794,825809,1075175
BC00224=126079,823643,1075175
BC00225=130858,823659,1075175
BC00226=170108,823795,1075173
BC00227=157966,823650,1075175
BC00228=156869,825691,1075175
BC00229=154126,830791,1075175
BC00230=114692,901690,1075175
BC00231=143002,931232,1075175
BC00232=146315,936443,1075175
BC00233=147641,938527,1075175
BC00234=194941,944470,1075175
BC00235=156841,937856,1075175
BC00236=172703,940853,1075175
BC00237=174292,939117,1075175
BC00238=178267,934778,1075175
BC00239=164918,911333,1075175
BC00240=91107,849480,1075175
BC00241=59698,829503,1075175
BC00242=57257,824323,1075175
BC00243=56280,822250,1075175
BC00244=29836,827677,1075175
BC00245=76754,827839,1075175
BC00246=27687,817329,1075175
BC00247=25853,819104,1075175
BC00248=21269,823543,1075175
BC00249=34689,834409,1075171
BC00250=267738,1017378,1075175
BC00251=272730,1015553,1075175
BC00252=274727,1014823,1075175
BC00253=328708,1053146,1075175
BC00254=294162,1033751,1075175
BC00255=279435,1024890,1075175
BC00256=269339,1011255,1075175
BC00257=265430,994958,1075175
BC00258=267336,981721,1075175
BC00259=271332,972471,1075175
BC00260=275026,965943,1075175
BC00261=277522,963553,1075175
BC00262=275862,962700,1075175
BC00263=272541,960996,1075175
BC00264=271715,892373,1073460
BC00265=294826,916334,1075175
BC00266=293545,921932,1075175
BC00267=293032,924172,1075175
BC00268=307043,929007,1075175
BC00269=302586,932369,1075175
BC00270=285695,927618,1075175
BC00271=319756,944028,1075175
BC00272=321000,944625,1075175
BC00273=321000,944625,1075175
BC00274=321000,944625,1075175
BC00275=325770,944528,1075175
BC00276=326754,940227,1075175
BC00277=126179,666204,1075175
BC00278=216726,717474,641306
BC00279=301368,789553,152612
BC00280=301368,789553,152612
BC00281=301368,789553,152612
BC00282=301368,789553,152612
BC00283=301368,789553,152612
BC00284=301368,789553,152612
BC00285=301368,789553,152612
BC00286=301368,789553,152612
BC00287=301368,789553,152612
BC00288=301368,789553,152612
BC00289=314485,789553,143111
BC00290=314485,789553,143111
BC00291=314485,789553,143111
BC00292=314485,789553,143111
BC00293=314485,789553,143111
BC00294=314485,789553,143111
BC00295=314485,789553,143111
BC00296=314485,789553,143111
BC00297=314485,789553,143111
BC00298=314485,789553,143111
BC00299=331615,789553,138281
BC00300=360333,789553,130184
BC00301=360333,789553,130184
BC00302=360333,789553,130184
BC00303=360333,789553,130184
BC00304=360333,789553,130184
BC00305=360333,789553,130184
BC00306=360333,789553,130184
BC00307=360333,789553,130184
BC00308=360333,789553,130184
BC00309=360333,789553,130184
BC00310=360333,789553,130184
BC00311=360105,789553,124885
BC00312=360105,789553,124885
BC00313=360106,789553,124884
BC00314=360106,789553,124884
BC00315=360106,789553,124884
BC00316=360106,789553,124884
BC00317=360106,789553,124884
BC00318=360105,789553,124885
BC00319=360105,789553,124885
BC00320=345851,783755,200789
BC00321=345851,783755,200789
BC00322=345851,783755,200789
BC00323=345851,783755,200789
BC00324=345851,783755,200789
BC00325=345851,783755,200789
BC00326=345851,783755,200789
BC00327=345851,783755,200789
BC00328=345851,783755,200789
BC00329=345851,783755,200789
BC00330=345851,783755,200789
BC00331=345851,783755,200789
BC00332=345851,783755,200789
BC00333=319787,789553,203514
BC00334=319787,789553,203514
BC00335=319787,790681,204440
BC00336=319787,790681,204440
BC00337=319787,790681,204440
BC00338=319787,790681,204440
BC00339=319787,790681,204440
BC00340=319787,790681,204440
BC00341=319787,790681,204440
BC00342=319787,790681,204440
BC00343=319787,790681,204440
BC00344=319787,790681,204440
BC00345=319787,790681,204440
BC00346=319787,790681,204440
BC00347=319787,790681,204440
BC00348=319787,790681,204440
BC00349=345989,790681,139065
BC00350=345989,790681,139065
BC00351=345988,790681,139065
BC00352=345988,790681,139065
BC00353=345988,790681,139065
BC00354=345988,790681,139065
BC00355=345988,790681,139065
BC00356=345988,790681,139065
BC00357=345988,790681,139065
BC00358=345988,790681,139065
BC00359=345988,790681,139065
BC00360=345988,790681,139065
BC00361=345988,790681,139065
BC00362=345988,790681,139065
BC00363=345988,790681,139065
BC00364=345989,790681,139065
BC00365=365235,789553,136516
BC00366=365235,789553,136516
BC00367=365235,789553,136514
BC00368=365235,789553,136514
BC00369=365235,789553,136514
BC00370=365235,789553,136514
BC00371=365235,789553,136514
BC00372=365235,789553,136516
BC00373=365235,789553,136516
BC00374=365235,669876,311777
BC00375=219200,669876,311777
BC00376=202290,739783,276486
BC00377=196160,765124,263693
BC00378=196160,765124,263693
BC00379=196160,765129,264619
BC00380=196160,765129,264619
BC00381=196160,765129,264619
BC00382=196160,765129,264619
BC00383=196160,765129,264619
BC00384=196160,765129,264619
BC00385=196160,765129,264619
BC00386=196160,765129,264619
BC00387=196160,765129,264619
BC00388=196160,765129,264619
BC00389=196160,765129,264619
BC00390=196160,765129,264619
BC00391=196160,765129,264619
BC00392=196160,765129,264619
BC00393=172117,778418,210988
BC00394=172117,778418,210988
BC00395=172117,778418,210988
BC00396=172117,778418,210988
BC00397=172117,778418,210988
BC00398=172117,778418,210988
BC00399=172117,778418,210988
BC00400=172117,778418,210988
BC00401=172117,778418,210988
BC00402=172117,778418,210988
BC00403=172117,778418,210988
BC00404=172117,778418,210988
BC00405=172117,778418,210988
BC00406=172117,778418,210988
BC00407=172117,778418,210988
BC00408=172117,778418,210988
BC00409=202290,739783,276486
BC00410=219200,669876,311777
BC00411=365235,669876,311777
BC00412=365235,789553,136516
BC00413=312307,789553,228155
BC00414=312307,789553,228155
BC00415=312307,789553,228155
BC00416=312307,789553,228155
BC00417=312307,789553,228155
BC00418=312307,789553,228155
BC00419=312307,789553,228155
BC00420=312307,789553,228155
BC00421=312307,789553,228155
BC00422=312307,789553,228155
BC00423=312307,789553,228155
BC00424=312307,789553,228155
BC00425=312307,789553,228155
BC00426=312307,789553,228155
BC00427=312307,789553,228155
BC00428=312307,789553,228155
BC00429=312307,789553,228155
BC00430=315278,774952,138157
BC00431=315278,774952,138157
BC00432=315278,774952,138157
BC00433=315278,774952,138157
BC00434=315278,774952,138157
BC00435=315278,774952,138157
BC00436=315278,774952,138157
BC00437=349744,788873,128099
BC00438=349744,788873,128099
BC00439=349744,788873,128099
BC00440=349744,788873,128099
BC00441=349744,788873,128099
BC00442=349744,788873,128099
BC00443=349744,788873,128099
BC00444=382626,789553,75740
BC00445=382626,789553,75740
BC00446=382625,789552,75737
BC00447=382625,789552,75737
BC00448=382626,789553,75740
BC00449=382626,789553,75740
BC00450=357624,789553,120797
BC00451=357624,789553,120797
BC00452=357624,789553,120797
BC00453=357624,789553,120797
BC00454=357624,789553,120797
BC00455=357624,789553,120797
BC00456=322012,789553,130156
BC00457=296072,789553,136973
BC00458=296072,789553,136973
BC00459=296072,789553,136973
BC00460=296072,789553,136973
BC00461=296072,789553,136973
BC00462=296072,789553,136973
BC00463=317007,789553,149819
BC00464=317007,789553,149819
BC00465=317007,789553,149819
BC00466=317007,789553,149819
BC00467=317007,789553,149819
BC00468=317007,789553,149819
BC00469=322972,789553,141208
BC00470=322972,789553,141208
BC00471=322972,789553,141208
BC00472=322972,789553,141208
BC00473=322972,789553,141208
BC00474=322972,789553,141208
BC00475=322972,668461,141208
BC00476=182890,668461,141208
BC00477=138897,773188,238096
BC00478=138897,773188,238096
BC00479=138897,773188,238096
BC00480=138897,773188,238096
BC00481=138897,773188,238096
BC00482=138897,773188,238096
BC00483=210738,761007,251818
BC00484=210738,761007,251818
BC00485=210738,761007,251818
BC00486=210738,761007,251818
BC00487=210738,761007,251818
BC00488=210738,761007,251818
BC00489=187715,774579,182649
BC00490=187715,774579,182649
BC00491=187715,774579,182649
BC00492=187715,774579,182649
BC00493=187715,774579,182649
BC00494=187715,774579,182649
BC00495=187905,774497,182612
BC00496=187905,774497,182612
BC00497=187905,774497,182612
BC00498=187905,774497,182612
BC00499=187905,774497,182612
BC00500=187905,774497,182612
BC00501=182890,668461,141208
BC00502=322972,668461,141208
BC00503=380287,789553,141173
BC00504=380287,789553,141173
BC00505=380287,789553,141173
BC00506=380287,789553,141173
BC00507=380287,789553,141173
BC00508=380287,789553,141173
BC00509=371434,789553,120731
BC00510=371434,789553,120731
BC00511=371434,789553,120731
BC00512=371434,789553,120731
BC00513=371434,789553,120731
BC00514=371434,789553,120731
BC00515=371434,685314,120731
BC00516=165820,667836,534036
EC00000=798156,0
EC00001=798156,0
EC00002=798156,0
EC00003=798156,0
EC00004=798156,0
EC00005=798156,0
EC00006=798156,0
EC00007=798156,0
EC00008=798156,0
EC00009=798156,0
EC00010=798156,0
EC00011=798156,0
EC00012=798156,0
EC00013=798156,0
EC00014=798156,0
EC00015=798156,0
EC00016=798156,0
EC00017=798156,0
EC00018=798156,0
EC00019=798156,0
EC00020=798156,0
EC00021=798156,0
EC00022=798156,0
EC00023=798156,0
EC00024=798156,0
EC00025=798156,0
EC00026=798156,0
EC00027=798156,0
EC00028=798156,0
EC00029=798156,0
EC00030=798156,0
EC00031=798156,0
EC00032=798156,0
EC00033=798156,0
EC00034=798156,0
EC00035=798156,0
EC00036=798156,0
EC00037=798156,0
EC00038=798156,0
EC00039=798156,0
EC00040=798156,0
EC00041=798156,0
EC00042=798156,0
EC00043=798156,0
EC00044=798156,0
EC00045=798156,0
EC00046=798156,0
EC00047=798156,0
EC00048=798156,0
EC00049=798156,0
EC00050=798156,0
EC00051=798156,0
EC00052=798156,0
EC00053=798156,0
EC00054=798156,0
EC00055=798156,0
EC00056=798156,0
EC00057=798156,0
EC00058=798156,0
EC00059=798156,0
EC00060=798156,0
EC00061=798156,0
EC00062=798156,0
EC00063=798156,0
EC00064=798156,0
EC00065=798156,0
EC00066=798156,0
EC00067=798156,0
EC00068=798156,0
EC00069=798156,0
EC00070=798156,0
EC00071=798156,0
EC00072=798156,0
EC00073=798156,0
EC00074=798156,0
EC00075=798156,0
EC00076=798156,0
EC00077=798156,0
EC00078=798156,0
EC00079=798156,0
EC00080=798156,0
EC00081=798156,0
EC00082=798156,0
EC00083=798156,0
EC00084=798156,0
EC00085=798156,0
EC00086=798156,0
EC00087=798156,0
EC00088=798156,0
EC00089=798156,0
EC00090=798156,0
EC00091=798156,0
EC00092=798156,0
EC00093=798156,0
EC00094=798156,0
EC00095=798156,0
EC00096=798156,0
EC00097=798156,0
EC00098=798156,0
EC00099=798156,0
EC00100=798156,0
EC00101=798156,0
EC00102=798156,0
EC00103=798156,0
EC00104=798156,0
EC00105=798156,0
EC00106=798156,0
EC00107=798156,0
EC00108=798156,0
EC00109=798156,0
EC00110=798156,0
EC00111=798156,0
EC00112=798156,0
EC00113=798156,0
EC00114=798156,0
EC00115=798156,0
EC00116=798156,0
EC00117=798156,0
EC00118=798156,0
EC00119=798156,0
EC00120=798156,0
EC00121=798156,0
EC00122=798156,0
EC00123=798156,0
EC00124=798156,0
EC00125=798156,0
EC00126=798156,0
EC00127=798156,0
EC00128=798156,0
EC00129=798156,0
EC00130=798156,0
EC00131=798156,0
EC00132=798156,0
EC00133=798156,0
EC00134=798156,0
EC00135=798156,0
EC00136=798156,0
EC00137=798156,0
EC00138=798156,0
EC00139=798156,0
EC00140=798156,0
EC00141=798156,0
EC00142=798156,0
EC00143=798156,0
EC00144=798156,0
EC00145=798156,0
EC00146=798156,0
EC00147=798156,0
EC00148=798156,0
EC00149=798156,0
EC00150=798156,0
EC00151=798156,0
EC00152=798156,0
EC00153=798156,0
EC00154=798156,0
EC00155=798156,0
EC00156=798156,0
EC00157=798156,0
EC00158=798156,0
EC00159=798156,0
EC00160=798156,0
EC00161=798156,0
EC00162=798156,0
EC00163=798156,0
EC00164=798156,0
EC00165=798156,0
EC00166=798156,0
EC00167=798156,0
EC00168=798156,0
EC00169=798156,0
EC00170=798156,0
EC00171=798156,0
EC00172=798156,0
EC00173=798155,0
EC00174=798155,1
EC00175=798155,0
EC00176=798155,1
EC00177=798156,0
EC00178=798156,0
EC00179=798156,0
EC00180=798156,0
EC00181=798156,0
EC00182=798156,0
EC00183=798156,0
EC00184=798156,0
EC00185=798156,0
EC00186=798156,0
EC00187=798156,0
EC00188=798156,0
EC00189=798156,0
EC00190=798156,0
EC00191=798156,0
EC00192=798156,0
EC00193=798153,3
EC00194=798156,0
EC00195=798156,0
EC00196=798156,0
EC00197=798156,0
EC00198=798156,0
EC00199=798156,0
EC00200=798156,0
EC00201=798156,0
EC00202=798156,0
EC00203=798156,0
EC00204=798156,0
EC00205=798156,0
EC00206=798155,0
EC00207=798156,0
EC00208=798156,0
EC00209=798156,0
EC00210=798156,0
EC00211=798156,0
EC00212=798156,0
EC00213=798156,0
EC00214=798156,0
EC00215=798156,0
EC00216=798156,0
EC00217=798156,0
EC00218=798156,0
EC00219=798156,0
EC00220=798156,0
EC00221=798156,0
EC00222=798156,0
EC00223=798156,0
EC00224=798156,0
EC00225=798156,0
EC00226=798155,0
EC00227=798156,0
EC00228=798156,0
EC00229=798156,0
EC00230=798156,0
EC00231=798156,0
EC00232=798156,0
EC00233=798156,0
EC00234=798156,0
EC00235=798156,0
EC00236=798156,0
EC00237=798156,0
EC00238=798156,0
EC00239=798156,0
EC00240=798156,0
EC00241=798156,0
EC00242=798156,0
EC00243=798156,0
EC00244=798156,0
EC00245=798156,0
EC00246=798156,0
EC00247=798156,0
EC00248=798156,0
EC00249=798155,0
EC00250=798156,0
EC00251=798156,0
EC00252=798156,0
EC00253=798156,0
EC00254=798156,0
EC00255=798156,0
EC00256=798156,0
EC00257=798156,0
EC00258=798156,0
EC00259=798156,0
EC00260=798156,0
EC00261=798156,0
EC00262=798156,0
EC00263=798156,0
EC00264=798156,0
EC00265=798156,0
EC00266=798156,0
EC00267=798156,0
EC00268=798156,0
EC00269=798156,0
EC00270=798156,0
EC00271=798156,0
EC00272=798156,0
EC00273=798156,0
EC00274=798156,0
EC00275=798156,0
EC00276=798156,0
EC00277=798156,0
EC00278=798156,0
EC00279=798156,0
EC00280=798156,0
EC00281=798156,0
EC00282=798156,0
EC00283=798156,0
EC00284=798156,0
EC00285=798156,0
EC00286=798156,0
EC00287=798156,0
EC00288=798156,0
EC00289=798156,0
EC00290=798156,0
EC00291=798156,0
EC00292=798156,0
EC00293=798156,0
EC00294=798156,0
EC00295=798156,0
EC00296=798156,0
EC00297=798156,0
EC00298=798156,0
EC00299=798156,0
EC00300=798156,0
EC00301=798156,0
EC00302=798156,0
EC00303=798156,0
EC00304=798156,0
EC00305=798156,0
EC00306=798156,0
EC00307=798156,0
EC00308=798156,0
EC00309=798156,0
EC00310=798156,0
EC00311=798156,0
EC00312=798156,0
EC00313=798156,1
EC00314=798156,1
EC00315=798156,1
EC00316=798156,1
EC00317=798156,1
EC00318=798156,0
EC00319=798156,0
EC00320=798156,0
EC00321=798156,0
EC00322=798156,0
EC00323=798156,0
EC00324=798156,0
EC00325=798156,0
EC00326=798156,0
EC00327=798156,0
EC00328=798156,0
EC00329=798156,0
EC00330=798156,0
EC00331=798156,0
EC00332=798156,0
EC00333=798156,0
EC00334=798156,0
EC00335=798156,0
EC00336=798156,0
EC00337=798156,0
EC00338=798156,0
EC00339=798156,0
EC00340=798156,0
EC00341=798156,0
EC00342=798156,0
EC00343=798156,0
EC00344=798156,0
EC00345=798156,0
EC00346=798156,0
EC00347=798156,0
EC00348=798156,0
EC00349=798156,0
EC00350=798156,0
EC00351=798156,1
EC00352=798156,1
EC00353=798156,1
EC00354=798156,1
EC00355=798156,1
EC00356=798156,1
EC00357=798156,1
EC00358=798156,1
EC00359=798156,1
EC00360=798156,1
EC00361=798156,1
EC00362=798156,1
EC00363=798156,1
EC00364=798156,0
EC00365=798156,0
EC00366=798156,0
EC00367=798155,1
EC00368=798155,1
EC00369=798155,1
EC00370=798155,1
EC00371=798155,1
EC00372=798156,0
EC00373=798156,0
EC00374=798156,0
EC00375=798156,0
EC00376=798156,0
EC00377=798156,0
EC00378=798156,0
EC00379=798156,0
EC00380=798156,0
EC00381=798156,0
EC00382=798156,0
EC00383=798156,0
EC00384=798156,0
EC00385=798156,0
EC00386=798156,0
EC00387=798156,0
EC00388=798156,0
EC00389=798156,0
EC00390=798156,0
EC00391=798156,0
EC00392=798156,0
EC00393=798156,0
EC00394=798156,0
EC00395=798156,0
EC00396=798156,0
EC00397=798156,0
EC00398=798156,0
EC00399=798156,0
EC00400=798156,0
EC00401=798156,0
EC00402=798156,0
EC00403=798156,0
EC00404=798156,0
EC00405=798156,0
EC00406=798156,0
EC00407=798156,0
EC00408=798156,0
EC00409=798156,0
EC00410=798156,0
EC00411=798156,0
EC00412=798156,0
EC00413=798156,0
EC00414=798156,0
EC00415=798156,0
EC00416=798156,0
EC00417=798156,0
EC00418=798156,0
EC00419=798156,0
EC00420=798156,0
EC00421=798156,0
EC00422=798156,0
EC00423=798156,0
EC00424=798156,0
EC00425=798156,0
EC00426=798156,0
EC00427=798156,0
EC00428=798156,0
EC00429=798156,0
EC00430=798156,0
EC00431=798156,0
EC00432=798156,0
EC00433=798156,0
EC00434=798156,0
EC00435=798156,0
EC00436=798156,0
EC00437=798156,0
EC00438=798156,0
EC00439=798156,0
EC00440=798156,0
EC00441=798156,0
EC00442=798156,0
EC00443=798156,0
EC00444=798156,0
EC00445=798156,0
EC00446=798155,0
EC00447=798155,0
EC00448=798156,0
EC00449=798156,0
EC00450=798156,0
EC00451=798156,0
EC00452=798156,0
EC00453=798156,0
EC00454=798156,0
EC00455=798156,0
EC00456=798156,0
EC00457=798156,0
EC00458=798156,0
EC00459=798156,0
EC00460=798156,0
EC00461=798156,0
EC00462=798156,0
EC00463=798156,0
EC00464=798156,0
EC00465=798156,0
EC00466=798156,0
EC00467=798156,0
EC00468=798156,0
EC00469=798156,0
EC00470=798156,0
EC00471=798156,0
EC00472=798156,0
EC00473=798156,0
EC00474=798156,0
EC00475=798156,0
EC00476=798156,0
EC00477=798156,0
EC00478=798156,0
EC00479=798156,0
EC00480=798156,0
EC00481=798156,0
EC00482=798156,0
EC00483=798156,0
EC00484=798156,0
EC00485=798156,0
EC00486=798156,0
EC00487=798156,0
EC00488=798156,0
EC00489=798156,0
EC00490=798156,0
EC00491=798156,0
EC00492=798156,0
EC00493=798156,0
EC00494=798156,0
EC00495=798156,0
EC00496=798156,0
EC00497=798156,0
EC00498=798156,0
EC00499=798156,0
EC00500=798156,0
EC00501=798156,0
EC00502=798156,0
EC00503=798156,0
EC00504=798156,0
EC00505=798156,0
EC00506=798156,0
EC00507=798156,0
EC00508=798156,0
EC00509=798156,0
EC00510=798156,0
EC00511=798156,0
EC00512=798156,0
EC00513=798156,0
EC00514=798156,0
EC00515=798156,0
EC00516=798156,0
///POSTYPE BASE
///RECTAN
///RCONF 0,0,0,0,0,0,0,0,0,0,0,0,0,0,0,0,0,0,0,0,0,0,0,0
P00006=0.222,-3.123,-1.508,0.0000,0.0000,0.0000
P00021=-0.225,-6.128,-0.405,0.0000,0.0000,0.0000
P00022=0.222,-3.123,-1.508,0.0000,0.0000,0.0000
P00023=0.143,-0.036,0.682,0.0000,0.0000,0.0000
P00024=0.145,-0.552,1.326,0.0000,0.0000,0.0000
P00025=-2.003,0.006,0.728,0.0000,0.0000,0.0000
P00026=0.562,-0.002,-0.337,0.0000,0.0000,0.0000
P00027=-0.746,0.015,-9.096,0.0000,0.0000,0.0000
P00028=-2.237,-0.018,-7.702,0.0000,0.0000,0.0000
P00029=-2.156,-0.086,-4.681,0.0000,0.0000,0.0000
P00030=5.926,-4.294,-1.390,0.0000,0.0000,0.0000
P00031=1.853,-0.001,-1.549,0.0000,0.0000,0.0000
P00032=1.957,0.503,-7.217,0.0000,0.0000,0.0000
///RCONF 0,0,0,0,1,0,0,0,0,0,0,0,0,0,0,0,0,0,0,0,0,0,0,0
P00033=-0.123,0.612,-5.012,0.0000,0.0000,0.0000
///RCONF 0,0,0,0,0,0,0,0,0,0,0,0,0,0,0,0,0,0,0,0,0,0,0,0
P00034=-0.304,0.773,-2.693,0.0000,0.0000,0.0000
P00042=-0.217,1.941,0.413,0.0000,0.0000,0.0000
P00043=-0.044,-1.937,1.197,0.0000,0.0000,0.0000
P00044=0.687,-2.322,1.156,0.0000,0.0000,0.0000
P00045=-0.068,-0.810,1.603,0.0000,0.0000,0.0000
P00046=0.799,0.043,1.292,0.0000,0.0000,0.0000
///RCONF 0,1,0,0,0,0,0,0,0,0,0,0,0,0,0,0,0,0,0,0,0,0,0,0
P00047=-0.011,1.737,-0.646,0.0000,0.0000,0.0000
///RCONF 0,0,0,0,0,0,0,0,0,0,0,0,0,0,0,0,0,0,0,0,0,0,0,0
P00048=2.411,0.025,-0.606,0.0000,0.0000,0.0000
P00049=3.413,-3.572,-1.618,0.0000,0.0000,0.0000
P00050=4.296,-4.501,-0.826,0.0000,0.0000,0.0000
P00051=0.367,3.892,0.009,0.0000,0.0000,0.0000
P00052=0.088,2.832,-0.342,0.0000,0.0000,0.0000
P00053=0.134,6.594,0.107,0.0000,0.0000,0.0000
P00054=-0.103,6.509,-0.702,0.0000,0.0000,0.0000
P00055=-0.342,8.912,1.324,0.0000,0.0000,0.0000
P00060=2.327,-2.514,-2.692,0.0000,0.0000,0.0000
P00091=-0.109,0.052,-0.075,0.0000,0.0000,0.0000
//INST
///DATE 2025/03/12 10:32
///ATTR SC,RW
///GROUP1 RB1,BS1
///GROUP2 ST1
NOP
'X2_38-47,64(2)(90,0)
'Down
MOVJ C00000 BC00000 VJ=100.00  +MOVJ EC00000 VJ=100.00
'Up
'Path S4602
SFTOF3D
COMM MOVJ C00001 BC00001 VJ=100.00  +MOVJ EC00001 VJ=100.00
COMM MOVL C00002 BC00002 V=800.0  +MOVJ EC00002 VJ=100.00
COMM SMOVL C00003 BC00003 V=166.7  +MOVJ EC00003
COMM SREFP 3 C00004 BC00004  +REFP EC00004
COMM CALL JOB:SEARCH-R1-S13D
COMM SET P021 P006
COMM SFTON3D P021
COMM SMOVL C00005 BC00005 V=166.7  +MOVJ EC00005
COMM SREFP 3 C00006 BC00006  +REFP EC00006
COMM CALL JOB:SEARCH-R1-S13D
COMM SET P021 P006
COMM SFTON3D P021
COMM SMOVL C00007 BC00007 V=166.7  +MOVJ EC00007
COMM MOVL C00008 BC00008 V=1000.0  +MOVJ EC00008 VJ=100.00
COMM 'EndPath S4602
COMM 'Path S4603
COMM SFTOF3D
COMM MOVJ C00009 BC00009 VJ=100.00  +MOVJ EC00009 VJ=100.00
COMM MOVL C00010 BC00010 V=800.0  +MOVJ EC00010 VJ=100.00
COMM SMOVL C00011 BC00011 V=166.7  +MOVJ EC00011
COMM SREFP 3 C00012 BC00012  +REFP EC00012
COMM CALL JOB:SEARCH-R1-S13D
COMM SET P022 P006
COMM SFTON3D P022
COMM SMOVL C00013 BC00013 V=166.7  +MOVJ EC00013
COMM SREFP 3 C00014 BC00014  +REFP EC00014
COMM CALL JOB:SEARCH-R1-S13D
COMM SET P022 P006
COMM SFTON3D P022
COMM SMOVL C00015 BC00015 V=166.7  +MOVJ EC00015
COMM MOVL C00016 BC00016 V=1000.0  +MOVJ EC00016 VJ=100.00
COMM 'EndPath S4603
COMM 'Path S4604
COMM SFTOF3D
MOVJ C00017 BC00017 VJ=100.00  +MOVJ EC00017 VJ=100.00
MOVJ C00018 BC00018 VJ=100.00  +MOVJ EC00018 VJ=100.00
MOVL C00019 BC00019 V=800.0  +MOVJ EC00019 VJ=100.00
SMOVL C00020 BC00020 V=166.7  +MOVJ EC00020
SREFP 3 C00021 BC00021  +REFP EC00021
CALL JOB:SEARCH-R1-S13D
SET P023 P006
SFTON3D P023
SMOVL C00022 BC00022 V=166.7  +MOVJ EC00022
SREFP 3 C00023 BC00023  +REFP EC00023
CALL JOB:SEARCH-R1-S13D
SET P023 P006
SFTON3D P023
SMOVL C00024 BC00024 V=166.7  +MOVJ EC00024
SMOVL C00025 BC00025 V=333.3  +MOVJ EC00025
SMOVL C00026 BC00026 V=333.3  +MOVJ EC00026
SREFP 3 C00027 BC00027  +REFP EC00027
CALL JOB:SEARCH-R1-S13D
SET P023 P006
SFTON3D P023
SMOVL C00028 BC00028 V=166.7  +MOVJ EC00028
MOVL C00029 BC00029 V=1000.0  +MOVJ EC00029 VJ=100.00
'EndPath S4604
'Path S4605
SFTOF3D
MOVJ C00030 BC00030 VJ=100.00  +MOVJ EC00030 VJ=100.00
MOVL C00031 BC00031 V=800.0  +MOVJ EC00031 VJ=100.00
SMOVL C00032 BC00032 V=166.7  +MOVJ EC00032
SREFP 3 C00033 BC00033  +REFP EC00033
CALL JOB:SEARCH-R1-S13D
SET P024 P006
SFTON3D P024
SMOVL C00034 BC00034 V=166.7  +MOVJ EC00034
SMOVL C00035 BC00035 V=166.7  +MOVJ EC00035
SREFP 3 C00036 BC00036  +REFP EC00036
CALL JOB:SEARCH-R1-S13D
SET P024 P006
SFTON3D P024
SMOVL C00037 BC00037 V=166.7  +MOVJ EC00037
SMOVL C00038 BC00038 V=166.7  +MOVJ EC00038
SREFP 3 C00039 BC00039  +REFP EC00039
CALL JOB:SEARCH-R1-S13D
SET P024 P006
SFTON3D P024
SMOVL C00040 BC00040 V=166.7  +MOVJ EC00040
MOVL C00041 BC00041 V=1000.0  +MOVJ EC00041 VJ=100.00
MOVL C00042 BC00042 V=1000.0  +MOVJ EC00042 VJ=100.00
'EndPath S4605
'Path S4606
SFTOF3D
MOVJ C00043 BC00043 VJ=100.00  +MOVJ EC00043 VJ=100.00
MOVL C00044 BC00044 V=800.0  +MOVJ EC00044 VJ=100.00
SMOVL C00045 BC00045 V=166.7  +MOVJ EC00045
SREFP 3 C00046 BC00046  +REFP EC00046
CALL JOB:SEARCH-R1-S13D
SET P025 P006
SFTON3D P025
SMOVL C00047 BC00047 V=166.7  +MOVJ EC00047
SREFP 3 C00048 BC00048  +REFP EC00048
CALL JOB:SEARCH-R1-S13D
SET P025 P006
SFTON3D P025
SMOVL C00049 BC00049 V=166.7  +MOVJ EC00049
SMOVL C00050 BC00050 V=166.7  +MOVJ EC00050
SREFP 3 C00051 BC00051  +REFP EC00051
CALL JOB:SEARCH-R1-S13D
SET P025 P006
SFTON3D P025
SMOVL C00052 BC00052 V=166.7  +MOVJ EC00052
MOVL C00053 BC00053 V=1000.0  +MOVJ EC00053 VJ=100.00
MOVL C00054 BC00054 V=1000.0  +MOVJ EC00054 VJ=100.00
'EndPath S4606
'Path S4607
SFTOF3D
MOVJ C00055 BC00055 VJ=100.00  +MOVJ EC00055 VJ=100.00
MOVL C00056 BC00056 V=800.0  +MOVJ EC00056 VJ=100.00
SMOVL C00057 BC00057 V=166.7  +MOVJ EC00057
SREFP 3 C00058 BC00058  +REFP EC00058
CALL JOB:SEARCH-R1-S13D
SET P026 P006
SFTON3D P026
SMOVL C00059 BC00059 V=166.7  +MOVJ EC00059
SREFP 3 C00060 BC00060  +REFP EC00060
CALL JOB:SEARCH-R1-S13D
SET P026 P006
SFTON3D P026
SMOVL C00061 BC00061 V=166.7  +MOVJ EC00061
MOVL C00062 BC00062 V=1000.0  +MOVJ EC00062 VJ=100.00
SFTOF3D
SMOVL C00063 BC00063 V=166.7  +MOVJ EC00063
SREFP 3 C00064 BC00064  +REFP EC00064
CALL JOB:SEARCH-R1-S13D
SET P091 P006
SFTON3D P091
SMOVL C00065 BC00065 V=166.7  +MOVJ EC00065
SREFP 3 C00066 BC00066  +REFP EC00066
CALL JOB:SEARCH-R1-S13D
SET P091 P006
SFTON3D P091
SMOVL C00067 BC00067 V=166.7  +MOVJ EC00067
SMOVL C00068 BC00068 V=500.0  +MOVJ EC00068
'EndPath S4607
MOVJ C00069 BC00069 VJ=100.00  +MOVJ EC00069 VJ=100.00
MOVJ C00070 BC00070 VJ=100.00  +MOVJ EC00070 VJ=100.00
'Path S4608
SFTOF3D
MOVJ C00071 BC00071 VJ=100.00  +MOVJ EC00071 VJ=100.00
MOVL C00072 BC00072 V=800.0  +MOVJ EC00072 VJ=100.00
SMOVL C00073 BC00073 V=166.7  +MOVJ EC00073
SREFP 3 C00074 BC00074  +REFP EC00074
CALL JOB:SEARCH-R1-S13D
SET P027 P006
SFTON3D P027
SMOVL C00075 BC00075 V=166.7  +MOVJ EC00075
SMOVL C00076 BC00076 V=166.7  +MOVJ EC00076
SREFP 3 C00077 BC00077  +REFP EC00077
CALL JOB:SEARCH-R1-S13D
SET P027 P006
SFTON3D P027
SMOVL C00078 BC00078 V=166.7  +MOVJ EC00078
SMOVL C00079 BC00079 V=166.7  +MOVJ EC00079
SREFP 3 C00080 BC00080  +REFP EC00080
CALL JOB:SEARCH-R1-S13D
SET P027 P006
SFTON3D P027
SMOVL C00081 BC00081 V=166.7  +MOVJ EC00081
MOVL C00082 BC00082 V=1000.0  +MOVJ EC00082 VJ=100.00
MOVL C00083 BC00083 V=1000.0  +MOVJ EC00083 VJ=100.00
'EndPath S4608
'Path S4609
SFTOF3D
MOVJ C00084 BC00084 VJ=100.00  +MOVJ EC00084 VJ=100.00
MOVL C00085 BC00085 V=800.0  +MOVJ EC00085 VJ=100.00
SMOVL C00086 BC00086 V=166.7  +MOVJ EC00086
SREFP 3 C00087 BC00087  +REFP EC00087
CALL JOB:SEARCH-R1-S13D
SET P028 P006
SFTON3D P028
SMOVL C00088 BC00088 V=166.7  +MOVJ EC00088
SREFP 3 C00089 BC00089  +REFP EC00089
CALL JOB:SEARCH-R1-S13D
SET P028 P006
SFTON3D P028
SMOVL C00090 BC00090 V=250.0  +MOVJ EC00090
MOVL C00091 BC00091 V=1000.0  +MOVJ EC00091 VJ=100.00
'EndPath S4609
MOVJ C00092 BC00092 VJ=100.00  +MOVJ EC00092 VJ=100.00
'Path S4882
SFTOF3D
MOVJ C00093 BC00093 VJ=100.00  +MOVJ EC00093 VJ=100.00
MOVL C00094 BC00094 V=800.0  +MOVJ EC00094 VJ=100.00
SMOVL C00095 BC00095 V=166.7  +MOVJ EC00095
SREFP 3 C00096 BC00096  +REFP EC00096
CALL JOB:SEARCH-R1-S13D
SET P060 P006
SFTON3D P060
SMOVL C00097 BC00097 V=166.7  +MOVJ EC00097
SMOVL C00098 BC00098 V=166.7  +MOVJ EC00098
SREFP 3 C00099 BC00099  +REFP EC00099
CALL JOB:SEARCH-R1-S13D
SET P060 P006
SFTON3D P060
SMOVL C00100 BC00100 V=166.7  +MOVJ EC00100
SMOVL C00101 BC00101 V=333.3  +MOVJ EC00101
SMOVL C00102 BC00102 V=166.7  +MOVJ EC00102
SREFP 3 C00103 BC00103  +REFP EC00103
CALL JOB:SEARCH-R1-S13D
SET P060 P006
SFTON3D P060
SMOVL C00104 BC00104 V=166.7  +MOVJ EC00104
MOVL C00105 BC00105 V=1000.0  +MOVJ EC00105 VJ=100.00
'EndPath S4882
MOVJ C00106 BC00106 VJ=100.00  +MOVJ EC00106 VJ=100.00
COMM 'Path S4610
COMM PAUSE
COMM SFTOF3D
COMM MOVJ C00107 BC00107 VJ=100.00  +MOVJ EC00107 VJ=100.00
COMM MOVL C00108 BC00108 V=800.0  +MOVJ EC00108 VJ=100.00
COMM SMOVL C00109 BC00109 V=166.7  +MOVJ EC00109
COMM SREFP 3 C00110 BC00110  +REFP EC00110
COMM CALL JOB:SEARCH-R1-S13D
COMM SET P029 P006
COMM SFTON3D P029
COMM SMOVL C00111 BC00111 V=166.7  +MOVJ EC00111
COMM SREFP 3 C00112 BC00112  +REFP EC00112
COMM CALL JOB:SEARCH-R1-S13D
COMM SET P029 P006
COMM SFTON3D P029
COMM SMOVL C00113 BC00113 V=166.7  +MOVJ EC00113
COMM MOVL C00114 BC00114 V=1000.0  +MOVJ EC00114 VJ=100.00
COMM 'EndPath S4610
COMM 'Path S4611
COMM SFTOF3D
COMM MOVJ C00115 BC00115 VJ=100.00  +MOVJ EC00115 VJ=100.00
COMM MOVL C00116 BC00116 V=800.0  +MOVJ EC00116 VJ=100.00
COMM SMOVL C00117 BC00117 V=166.7  +MOVJ EC00117
COMM SREFP 3 C00118 BC00118  +REFP EC00118
COMM CALL JOB:SEARCH-R1-S13D
COMM SET P030 P006
COMM SFTON3D P030
COMM SMOVL C00119 BC00119 V=166.7  +MOVJ EC00119
COMM SREFP 3 C00120 BC00120  +REFP EC00120
COMM CALL JOB:SEARCH-R1-S13D
COMM SET P030 P006
COMM SFTON3D P030
COMM SMOVL C00121 BC00121 V=166.7  +MOVJ EC00121
COMM MOVL C00122 BC00122 V=800.0  +MOVJ EC00122 VJ=100.00
COMM MOVL C00123 BC00123 V=1000.0  +MOVJ EC00123 VJ=100.00
COMM 'EndPath S4611
MOVJ C00124 BC00124 VJ=100.00  +MOVJ EC00124 VJ=100.00
'Path S4612
SFTOF3D
MOVJ C00125 BC00125 VJ=100.00  +MOVJ EC00125 VJ=100.00
MOVL C00126 BC00126 V=800.0  +MOVJ EC00126 VJ=100.00
SMOVL C00127 BC00127 V=166.7  +MOVJ EC00127
SREFP 3 C00128 BC00128  +REFP EC00128
CALL JOB:SEARCH-R1-S13D
SET P031 P006
SFTON3D P031
SMOVL C00129 BC00129 V=166.7  +MOVJ EC00129
SMOVL C00130 BC00130 V=166.7  +MOVJ EC00130
SREFP 3 C00131 BC00131  +REFP EC00131
CALL JOB:SEARCH-R1-S13D
SET P031 P006
SFTON3D P031
SMOVL C00132 BC00132 V=166.7  +MOVJ EC00132
SMOVL C00133 BC00133 V=166.7  +MOVJ EC00133
SREFP 3 C00134 BC00134  +REFP EC00134
CALL JOB:SEARCH-R1-S13D
SET P031 P006
SFTON3D P031
SMOVL C00135 BC00135 V=166.7  +MOVJ EC00135
MOVL C00136 BC00136 V=1000.0  +MOVJ EC00136 VJ=100.00
'EndPath S4612
MOVJ C00137 BC00137 VJ=100.00  +MOVJ EC00137 VJ=100.00
'Path S4613
SFTOF3D
MOVJ C00138 BC00138 VJ=100.00  +MOVJ EC00138 VJ=100.00
MOVL C00139 BC00139 V=800.0  +MOVJ EC00139 VJ=100.00
SMOVL C00140 BC00140 V=166.7  +MOVJ EC00140
SREFP 3 C00141 BC00141  +REFP EC00141
CALL JOB:SEARCH-R1-S13D
SET P032 P006
SFTON3D P032
SMOVL C00142 BC00142 V=166.7  +MOVJ EC00142
SREFP 3 C00143 BC00143  +REFP EC00143
CALL JOB:SEARCH-R1-S13D
SET P032 P006
SFTON3D P032
SMOVL C00144 BC00144 V=166.7  +MOVJ EC00144
SMOVL C00145 BC00145 V=166.7  +MOVJ EC00145
SREFP 3 C00146 BC00146  +REFP EC00146
CALL JOB:SEARCH-R1-S13D
SET P032 P006
SFTON3D P032
SMOVL C00147 BC00147 V=166.7  +MOVJ EC00147
MOVL C00148 BC00148 V=1000.0  +MOVJ EC00148 VJ=100.00
'EndPath S4613
MOVJ C00149 BC00149 VJ=100.00  +MOVJ EC00149 VJ=100.00
'Path S4614
SFTOF3D
MOVJ C00150 BC00150 VJ=100.00  +MOVJ EC00150 VJ=100.00
MOVL C00151 BC00151 V=800.0  +MOVJ EC00151 VJ=100.00
SMOVL C00152 BC00152 V=166.7  +MOVJ EC00152
SREFP 3 C00153 BC00153  +REFP EC00153
CALL JOB:SEARCH-R1-S13D
SET P033 P006
SFTON3D P033
SMOVL C00154 BC00154 V=166.7  +MOVJ EC00154
SREFP 3 C00155 BC00155  +REFP EC00155
CALL JOB:SEARCH-R1-S13D
SET P033 P006
SFTON3D P033
SMOVL C00156 BC00156 V=166.7  +MOVJ EC00156
MOVL C00157 BC00157 V=1000.0  +MOVJ EC00157 VJ=100.00
'EndPath S4614
'Path S4615
SFTOF3D
MOVJ C00158 BC00158 VJ=100.00  +MOVJ EC00158 VJ=100.00
MOVL C00159 BC00159 V=800.0  +MOVJ EC00159 VJ=100.00
SMOVL C00160 BC00160 V=166.7  +MOVJ EC00160
SREFP 3 C00161 BC00161  +REFP EC00161
CALL JOB:SEARCH-R1-S13D
SET P034 P006
SFTON3D P034
SMOVL C00162 BC00162 V=166.7  +MOVJ EC00162
SREFP 3 C00163 BC00163  +REFP EC00163
CALL JOB:SEARCH-R1-S13D
SET P034 P006
SFTON3D P034
SMOVL C00164 BC00164 V=166.7  +MOVJ EC00164
SMOVL C00165 BC00165 V=166.7  +MOVJ EC00165
SREFP 3 C00166 BC00166  +REFP EC00166
CALL JOB:SEARCH-R1-S13D
SET P034 P006
SFTON3D P034
SMOVL C00167 BC00167 V=166.7  +MOVJ EC00167
MOVL C00168 BC00168 V=1000.0  +MOVJ EC00168 VJ=100.00
'EndPath S4615
MOVJ C00169 BC00169 VJ=100.00  +MOVJ EC00169 VJ=100.00
MOVJ C00170 BC00170 VJ=100.00  +MOVJ EC00170 VJ=100.00
'Path W4616
SFTOF3D
SFTON3D P026
MOVJ C00171 BC00171 VJ=100.00  +MOVJ EC00171 VJ=100.00
SMOVL C00172 BC00172 V=800.0  +MOVJ EC00172
'POPRAWIC!!!!
SMOVL C00173 BC00173 V=166.7 PL=0  +MOVJ EC00173
MACRO1 MJ#(0) ARGF21
ARCON
SWVON WEV#(100)
SMOVL C00174 BC00174 V=9.2  +MOVJ EC00174
SFTON3D P091
SMOVL C00175 BC00175 V=9.2  +MOVJ EC00175
SMOVL C00176 BC00176 V=9.2  +MOVJ EC00176
SWVOF
ARCOF
SMOVL C00177 BC00177 V=800.0  +MOVJ EC00177
SMOVL C00178 BC00178 V=1000.0  +MOVJ EC00178
SFTOF3D
'EndPath W4616
MOVJ C00179 BC00179 VJ=100.00  +MOVJ EC00179 VJ=100.00
'Path W4617
SFTOF3D
SFTON3D P028
MOVJ C00180 BC00180 VJ=100.00  +MOVJ EC00180 VJ=100.00
MOVJ C00181 BC00181 VJ=100.00  +MOVJ EC00181 VJ=100.00
SMOVL C00182 BC00182 V=800.0  +MOVJ EC00182
SMOVL C00183 BC00183 V=150.0 PL=0  +MOVJ EC00183
ARCON
SWVON WEV#(100)
MOVL C00184 BC00184 V=9.2  +MOVJ EC00184 VJ=100.00
SFTON3D P027
SMOVL C00185 BC00185 V=9.2  +MOVJ EC00185
SMOVL C00186 BC00186 V=9.2  +MOVJ EC00186
ARCOF
SWVOF
SMOVL C00187 BC00187 V=800.0  +MOVJ EC00187
SMOVL C00188 BC00188 V=1000.0  +MOVJ EC00188
SFTOF3D
'EndPath W4617
MOVJ C00189 BC00189 VJ=100.00  +MOVJ EC00189 VJ=100.00
'Path W4618
COMM PAUSE
COMM SFTOF3D
COMM SFTON3D P022
COMM MOVJ C00190 BC00190 VJ=100.00  +MOVJ EC00190 VJ=100.00
COMM SMOVL C00191 BC00191 V=800.0  +MOVJ EC00191
COMM SMOVL C00192 BC00192 V=150.0 PL=0  +MOVJ EC00192
COMM MACRO1 MJ#(0) ARGF9
COMM ARCON
COMM SWVON WEV#(60)
COMM SFTON3D P021
COMM SMOVL C00193 BC00193 V=10.0  +MOVJ EC00193
COMM ARCOF
COMM SWVOF
COMM SMOVL C00194 BC00194 V=800.0  +MOVJ EC00194
COMM SMOVL C00195 BC00195 V=1000.0  +MOVJ EC00195
COMM SFTOF3D
COMM 'EndPath W4618
COMM 'Path W4883
SFTOF3D
SFTON3D P060
MOVJ C00196 BC00196 VJ=100.00  +MOVJ EC00196 VJ=100.00
MACRO1 MJ#(0) ARGF9
SMOVL C00197 BC00197 V=800.0  +MOVJ EC00197
SMOVL C00198 BC00198 V=150.0 PL=0  +MOVJ EC00198
ARCON
SMOVL C00199 BC00199 V=10.0  +MOVJ EC00199
SMOVL C00200 BC00200 V=10.0  +MOVJ EC00200
SMOVL C00201 BC00201 V=10.0  +MOVJ EC00201
ARCOF
SMOVL C00202 BC00202 V=800.0  +MOVJ EC00202
SFTOF3D
'EndPath W4883
'Path W4884
SFTOF3D
SFTON3D P060
SMOVL C00203 BC00203 V=800.0  +MOVJ EC00203
SMOVL C00204 BC00204 V=150.0 PL=0  +MOVJ EC00204
ARCON
SMOVL C00205 BC00205 V=10.0  +MOVJ EC00205
SMOVL C00206 BC00206 V=10.0  +MOVJ EC00206
SMOVL C00207 BC00207 V=10.0  +MOVJ EC00207
ARCOF
SMOVL C00208 BC00208 V=800.0  +MOVJ EC00208
SMOVL C00209 BC00209 V=1000.0  +MOVJ EC00209
SFTOF3D
'EndPath W4884
MOVJ C00210 BC00210 VJ=100.00  +MOVJ EC00210 VJ=100.00
COMM 'Path W4619
COMM PAUSE
COMM SFTOF3D
COMM SFTON3D P030
COMM MOVJ C00211 BC00211 VJ=100.00  +MOVJ EC00211 VJ=100.00
COMM MOVJ C00212 BC00212 VJ=100.00  +MOVJ EC00212 VJ=100.00
COMM SMOVL C00213 BC00213 V=800.0  +MOVJ EC00213
COMM SMOVL C00214 BC00214 V=150.0 PL=0  +MOVJ EC00214
COMM ARCON
COMM MOVL C00215 BC00215 V=10.0  +MOVJ EC00215 VJ=100.00
COMM SFTON3D P029
COMM SMOVL C00216 BC00216 V=10.0  +MOVJ EC00216
COMM SMOVL C00217 BC00217 V=10.0  +MOVJ EC00217
COMM ARCOF
COMM SMOVL C00218 BC00218 V=800.0  +MOVJ EC00218
COMM SMOVL C00219 BC00219 V=1000.0  +MOVJ EC00219
COMM SFTOF3D
COMM 'EndPath W4619
MOVJ C00220 BC00220 VJ=100.00  +MOVJ EC00220 VJ=100.00
MOVJ C00221 BC00221 VJ=100.00  +MOVJ EC00221 VJ=100.00
'Path W4620
SFTOF3D
SFTON3D P033
MOVJ C00222 BC00222 VJ=100.00  +MOVJ EC00222 VJ=100.00
SMOVL C00223 BC00223 V=800.0  +MOVJ EC00223
SMOVL C00224 BC00224 V=166.7 PL=0  +MOVJ EC00224
ARCON
SMOVL C00225 BC00225 V=9.2  +MOVJ EC00225
SFTON3D P034
SMOVL C00226 BC00226 V=9.2  +MOVJ EC00226
SMOVL C00227 BC00227 V=9.2  +MOVJ EC00227
ARCOF
SMOVL C00228 BC00228 V=800.0  +MOVJ EC00228
SMOVL C00229 BC00229 V=1000.0  +MOVJ EC00229
SFTOF3D
'EndPath W4620
MOVJ C00230 BC00230 VJ=100.00  +MOVJ EC00230 VJ=100.00
'Path W4621
SFTOF3D
SFTON3D P024
MOVJ C00231 BC00231 VJ=100.00  +MOVJ EC00231 VJ=100.00
SMOVL C00232 BC00232 V=800.0  +MOVJ EC00232
SMOVL C00233 BC00233 V=166.7 PL=0  +MOVJ EC00233
ARCON
SMOVL C00234 BC00234 V=10.0  +MOVJ EC00234
SFTON3D P025
SMOVL C00235 BC00235 V=10.0  +MOVJ EC00235
SMOVL C00236 BC00236 V=10.0  +MOVJ EC00236
ARCOF
SMOVL C00237 BC00237 V=800.0  +MOVJ EC00237
SMOVL C00238 BC00238 V=1000.0  +MOVJ EC00238
SFTOF3D
'EndPath W4621
MOVJ C00239 BC00239 VJ=100.00  +MOVJ EC00239 VJ=100.00
MOVJ C00240 BC00240 VJ=100.00  +MOVJ EC00240 VJ=100.00
'Path W4622
SFTOF3D
SFTON3D P032
MOVJ C00241 BC00241 VJ=100.00  +MOVJ EC00241 VJ=100.00
SMOVL C00242 BC00242 V=800.0  +MOVJ EC00242
SMOVL C00243 BC00243 V=166.7 PL=0  +MOVJ EC00243
ARCON
SMOVL C00244 BC00244 V=9.2  +MOVJ EC00244
SFTON3D P031
SMOVL C00245 BC00245 V=9.2  +MOVJ EC00245
SMOVL C00246 BC00246 V=9.2  +MOVJ EC00246
ARCOF
SMOVL C00247 BC00247 V=800.0  +MOVJ EC00247
SMOVL C00248 BC00248 V=1000.0  +MOVJ EC00248
SFTOF3D
'EndPath W4622
'Path W4623
SFTOF3D
SFTON3D P023
MOVJ C00249 BC00249 VJ=100.00  +MOVJ EC00249 VJ=100.00
JUMP *VVP
MOVJ C00250 BC00250 VJ=100.00  +MOVJ EC00250 VJ=100.00
SMOVL C00251 BC00251 V=800.0  +MOVJ EC00251
SMOVL C00252 BC00252 V=166.7 PL=0  +MOVJ EC00252
'ARCON DO SPRAWDZENIA
PAUSE
SMOVL C00253 BC00253 V=10.0  +MOVJ EC00253
SMOVL C00254 BC00254 V=10.0  +MOVJ EC00254
SMOVL C00255 BC00255 V=10.0  +MOVJ EC00255
SMOVL C00256 BC00256 V=10.0  +MOVJ EC00256
SMOVL C00257 BC00257 V=10.0  +MOVJ EC00257
SMOVL C00258 BC00258 V=10.0  +MOVJ EC00258
SMOVL C00259 BC00259 V=10.0  +MOVJ EC00259
SMOVL C00260 BC00260 V=10.0  +MOVJ EC00260
SMOVL C00261 BC00261 V=10.0  +MOVJ EC00261
ARCOF
SMOVL C00262 BC00262 V=800.0  +MOVJ EC00262
SMOVL C00263 BC00263 V=1000.0  +MOVJ EC00263
SFTOF3D
'EndPath W4623
'Path W4624
*VVP
MOVJ C00264 BC00264 VJ=100.00  +MOVJ EC00264 VJ=100.00
SFTOF3D
SFTON3D P023
MOVJ C00265 BC00265 VJ=100.00  +MOVJ EC00265 VJ=100.00
SMOVL C00266 BC00266 V=800.0  +MOVJ EC00266
COMM SMOVL C00267 BC00267 V=150.0 PL=0  +MOVJ EC00267
COMM ARCON
COMM SMOVL C00268 BC00268 V=8.3  +MOVJ EC00268
SMOVL C00269 BC00269 V=166.7 PL=0  +MOVJ EC00269
ARCON
SMOVL C00270 BC00270 V=8.3  +MOVJ EC00270
SMOVL C00271 BC00271 V=8.3  +MOVJ EC00271
SMOVL C00272 BC00272 V=8.3  +MOVJ EC00272
SMOVL C00273 BC00273 V=8.3  +MOVJ EC00273
MOVL C00274 BC00274 V=8.3  +MOVJ EC00274 VJ=100.00
ARCOF
SMOVL C00275 BC00275 V=800.0  +MOVJ EC00275
SMOVL C00276 BC00276 V=1000.0  +MOVJ EC00276
SFTOF3D
'EndPath W4624
MOVJ C00277 BC00277 VJ=100.00  +MOVJ EC00277 VJ=100.00
'Path S4625
SFTOF3D
CALL JOB:CLEAN-R1_KM_3P
MOVJ C00278 BC00278 VJ=100.00  +MOVJ EC00278 VJ=100.00
MOVJ C00279 BC00279 VJ=100.00  +MOVJ EC00279 VJ=100.00
MOVL C00280 BC00280 V=800.0  +MOVJ EC00280 VJ=100.00
SMOVL C00281 BC00281 V=166.7  +MOVJ EC00281
SREFP 3 C00282 BC00282  +REFP EC00282
CALL JOB:SEARCH-R1-S13D
SET P048 P006
SFTON3D P048
SMOVL C00283 BC00283 V=166.7  +MOVJ EC00283
SMOVL C00284 BC00284 V=166.7  +MOVJ EC00284
SREFP 3 C00285 BC00285  +REFP EC00285
CALL JOB:SEARCH-R1-S13D
SET P048 P006
SFTON3D P048
SMOVL C00286 BC00286 V=16.7  +MOVJ EC00286
MOVL C00287 BC00287 V=800.0  +MOVJ EC00287 VJ=100.00
MOVL C00288 BC00288 V=1000.0  +MOVJ EC00288 VJ=100.00
'EndPath S4625
'Path S4626
SFTOF3D
MOVJ C00289 BC00289 VJ=100.00  +MOVJ EC00289 VJ=100.00
MOVL C00290 BC00290 V=800.0  +MOVJ EC00290 VJ=100.00
SMOVL C00291 BC00291 V=166.7  +MOVJ EC00291
SREFP 3 C00292 BC00292  +REFP EC00292
CALL JOB:SEARCH-R1-S13D
SET P047 P006
SFTON3D P047
SMOVL C00293 BC00293 V=166.7  +MOVJ EC00293
SMOVL C00294 BC00294 V=166.7  +MOVJ EC00294
SREFP 3 C00295 BC00295  +REFP EC00295
CALL JOB:SEARCH-R1-S13D
SET P047 P006
SFTON3D P047
SMOVL C00296 BC00296 V=166.7  +MOVJ EC00296
MOVL C00297 BC00297 V=800.0  +MOVJ EC00297 VJ=100.00
MOVL C00298 BC00298 V=1000.0  +MOVJ EC00298 VJ=100.00
'EndPath S4626
MOVJ C00299 BC00299 VJ=100.00  +MOVJ EC00299 VJ=100.00
'Path S4627
SFTOF3D
MOVJ C00300 BC00300 VJ=100.00  +MOVJ EC00300 VJ=100.00
MOVL C00301 BC00301 V=800.0  +MOVJ EC00301 VJ=100.00
SMOVL C00302 BC00302 V=166.7  +MOVJ EC00302
SREFP 3 C00303 BC00303  +REFP EC00303
CALL JOB:SEARCH-R1-S13D
SET P046 P006
SFTON3D P046
SMOVL C00304 BC00304 V=166.7  +MOVJ EC00304
MOVL C00305 BC00305 V=800.0  +MOVJ EC00305 VJ=100.00
SMOVL C00306 BC00306 V=166.7  +MOVJ EC00306
SREFP 3 C00307 BC00307  +REFP EC00307
CALL JOB:SEARCH-R1-S13D
SET P046 P006
SFTON3D P046
SMOVL C00308 BC00308 V=166.7  +MOVJ EC00308
MOVL C00309 BC00309 V=800.0  +MOVJ EC00309 VJ=100.00
MOVL C00310 BC00310 V=1000.0  +MOVJ EC00310 VJ=100.00
'EndPath S4627
'Path S4628
SFTOF3D
MOVJ C00311 BC00311 VJ=100.00  +MOVJ EC00311 VJ=100.00
MOVL C00312 BC00312 V=800.0  +MOVJ EC00312 VJ=100.00
SMOVL C00313 BC00313 V=166.7  +MOVJ EC00313
SREFP 3 C00314 BC00314  +REFP EC00314
CALL JOB:SEARCH-R1-S13D
SET P050 P006
SFTON3D P050
SMOVL C00315 BC00315 V=166.7  +MOVJ EC00315
SREFP 3 C00316 BC00316  +REFP EC00316
CALL JOB:SEARCH-R1-S13D
SET P050 P006
SFTON3D P050
SMOVL C00317 BC00317 V=166.7  +MOVJ EC00317
MOVL C00318 BC00318 V=800.0  +MOVJ EC00318 VJ=100.00
MOVL C00319 BC00319 V=1000.0  +MOVJ EC00319 VJ=100.00
'EndPath S4628
'Path S4629
SFTOF3D
MOVJ C00320 BC00320 VJ=100.00  +MOVJ EC00320 VJ=100.00
MOVJ C00321 BC00321 VJ=100.00  +MOVJ EC00321 VJ=100.00
MOVL C00322 BC00322 V=800.0  +MOVJ EC00322 VJ=100.00
SMOVL C00323 BC00323 V=166.7  +MOVJ EC00323
SREFP 3 C00324 BC00324  +REFP EC00324
CALL JOB:SEARCH-R1-S13D
SET P051 P006
SFTON3D P051
SMOVL C00325 BC00325 V=166.7  +MOVJ EC00325
SREFP 3 C00326 BC00326  +REFP EC00326
CALL JOB:SEARCH-R1-S13D
SET P051 P006
SFTON3D P051
SMOVL C00327 BC00327 V=166.7  +MOVJ EC00327
SMOVL C00328 BC00328 V=250.0  +MOVJ EC00328
SMOVL C00329 BC00329 V=166.7  +MOVJ EC00329
SREFP 3 C00330 BC00330  +REFP EC00330
CALL JOB:SEARCH-R1-S13D
SET P051 P006
SFTON3D P051
SMOVL C00331 BC00331 V=166.7  +MOVJ EC00331
MOVL C00332 BC00332 V=1000.0  +MOVJ EC00332 VJ=100.00
'EndPath S4629
'Path S4630
SFTOF3D
MOVJ C00333 BC00333 VJ=100.00  +MOVJ EC00333 VJ=100.00
MOVL C00334 BC00334 V=800.0  +MOVJ EC00334 VJ=100.00
SMOVL C00335 BC00335 V=166.7  +MOVJ EC00335
SREFP 3 C00336 BC00336  +REFP EC00336
CALL JOB:SEARCH-R1-S13D
SET P055 P006
SFTON3D P055
SMOVL C00337 BC00337 V=166.7  +MOVJ EC00337
SMOVL C00338 BC00338 V=166.7  +MOVJ EC00338
SMOVL C00339 BC00339 V=166.7  +MOVJ EC00339
SREFP 3 C00340 BC00340  +REFP EC00340
CALL JOB:SEARCH-R1-S13D
SET P055 P006
SFTON3D P055
SMOVL C00341 BC00341 V=166.7  +MOVJ EC00341
SREFP 3 C00342 BC00342  +REFP EC00342
CALL JOB:SEARCH-R1-S13D
SET P045 P006
SFTON3D P045
SMOVL C00343 BC00343 V=166.7  +MOVJ EC00343
SMOVL C00344 BC00344 V=166.7  +MOVJ EC00344
SMOVL C00345 BC00345 V=166.7  +MOVJ EC00345
SREFP 3 C00346 BC00346  +REFP EC00346
CALL JOB:SEARCH-R1-S13D
SET P045 P006
SFTON3D P045
SMOVL C00347 BC00347 V=166.7  +MOVJ EC00347
MOVL C00348 BC00348 V=1000.0  +MOVJ EC00348 VJ=100.00
'EndPath S4007
'Path S3506
SFTOF3D
MOVJ C00349 BC00349 VJ=100.00  +MOVJ EC00349 VJ=100.00
MOVL C00350 BC00350 V=666.7  +MOVJ EC00350 VJ=100.00
MOVL C00351 BC00351 V=166.7  +MOVJ EC00351 VJ=0.78
SREFP 3 C00352 BC00352  +REFP EC00352
CALL JOB:SEARCH-R1-S13D
SET P054 P006
SFTON3D P054
SMOVL C00353 BC00353 V=166.7  +MOVJ EC00353
SMOVL C00354 BC00354 V=166.7  +MOVJ EC00354
SMOVL C00355 BC00355 V=166.7  +MOVJ EC00355
SREFP 3 C00356 BC00356  +REFP EC00356
CALL JOB:SEARCH-R1-S13D
SET P054 P006
SFTON3D P054
SMOVL C00357 BC00357 V=166.7  +MOVJ EC00357
SREFP 3 C00358 BC00358  +REFP EC00358
CALL JOB:SEARCH-R1-S13D
SET P044 P006
SFTON3D P044
SMOVL C00359 BC00359 V=166.7  +MOVJ EC00359
SMOVL C00360 BC00360 V=166.7  +MOVJ EC00360
SMOVL C00361 BC00361 V=166.7  +MOVJ EC00361
SREFP 3 C00362 BC00362  +REFP EC00362
CALL JOB:SEARCH-R1-S13D
SET P044 P006
SFTON3D P044
SMOVL C00363 BC00363 V=166.7  +MOVJ EC00363
MOVL C00364 BC00364 V=1000.0  +MOVJ EC00364 VJ=100.00
SFTOF3D
MOVJ C00365 BC00365 VJ=100.00  +MOVJ EC00365 VJ=100.00
MOVL C00366 BC00366 V=800.0  +MOVJ EC00366 VJ=100.00
SMOVL C00367 BC00367 V=166.7  +MOVJ EC00367
SREFP 3 C00368 BC00368  +REFP EC00368
CALL JOB:SEARCH-R1-S13D
SET P049 P006
SFTON3D P049
SMOVL C00369 BC00369 V=166.7  +MOVJ EC00369
SREFP 3 C00370 BC00370  +REFP EC00370
CALL JOB:SEARCH-R1-S13D
SET P049 P006
SFTON3D P049
SMOVL C00371 BC00371 V=166.7  +MOVJ EC00371
MOVL C00372 BC00372 V=1000.0  +MOVJ EC00372 VJ=100.00
'EndPath S4632
MOVJ C00373 BC00373 VJ=100.00  +MOVJ EC00373 VJ=100.00
MOVJ C00374 BC00374 VJ=100.00  +MOVJ EC00374 VJ=100.00
MOVJ C00375 BC00375 VJ=100.00  +MOVJ EC00375 VJ=100.00
MOVJ C00376 BC00376 VJ=100.00  +MOVJ EC00376 VJ=100.00
'Path S4633
SFTOF3D
MOVJ C00377 BC00377 VJ=100.00  +MOVJ EC00377 VJ=100.00
MOVL C00378 BC00378 V=800.0  +MOVJ EC00378 VJ=100.00
SMOVL C00379 BC00379 V=166.7  +MOVJ EC00379
SREFP 3 C00380 BC00380  +REFP EC00380
CALL JOB:SEARCH-R1-S13D
SET P053 P006
SFTON3D P053
SMOVL C00381 BC00381 V=166.7  +MOVJ EC00381
SMOVL C00382 BC00382 V=166.7  +MOVJ EC00382
SMOVL C00383 BC00383 V=166.7  +MOVJ EC00383
SREFP 3 C00384 BC00384  +REFP EC00384
CALL JOB:SEARCH-R1-S13D
SET P053 P006
SFTON3D P053
SMOVL C00385 BC00385 V=166.7  +MOVJ EC00385
SREFP 3 C00386 BC00386  +REFP EC00386
CALL JOB:SEARCH-R1-S13D
SET P043 P006
SFTON3D P043
SMOVL C00387 BC00387 V=166.7  +MOVJ EC00387
SMOVL C00388 BC00388 V=166.7  +MOVJ EC00388
SMOVL C00389 BC00389 V=166.7  +MOVJ EC00389
SREFP 3 C00390 BC00390  +REFP EC00390
CALL JOB:SEARCH-R1-S13D
SET P043 P006
SFTON3D P043
SMOVL C00391 BC00391 V=166.7  +MOVJ EC00391
MOVL C00392 BC00392 V=1000.0  +MOVJ EC00392 VJ=100.00
'EndPath S4006
'Path S4005
SFTOF3D
MOVJ C00393 BC00393 VJ=100.00  +MOVJ EC00393 VJ=100.00
MOVL C00394 BC00394 V=800.0  +MOVJ EC00394 VJ=100.00
SMOVL C00395 BC00395 V=166.7  +MOVJ EC00395
SREFP 3 C00396 BC00396  +REFP EC00396
CALL JOB:SEARCH-R1-S13D
SET P052 P006
SFTON3D P052
SMOVL C00397 BC00397 V=166.7  +MOVJ EC00397
SMOVL C00398 BC00398 V=166.7  +MOVJ EC00398
SMOVL C00399 BC00399 V=166.7  +MOVJ EC00399
SREFP 3 C00400 BC00400  +REFP EC00400
CALL JOB:SEARCH-R1-S13D
SET P052 P006
SFTON3D P052
SMOVL C00401 BC00401 V=166.7  +MOVJ EC00401
SREFP 3 C00402 BC00402  +REFP EC00402
CALL JOB:SEARCH-R1-S13D
SET P042 P006
SFTON3D P042
SMOVL C00403 BC00403 V=166.7  +MOVJ EC00403
SMOVL C00404 BC00404 V=166.7  +MOVJ EC00404
SMOVL C00405 BC00405 V=166.7  +MOVJ EC00405
SREFP 3 C00406 BC00406  +REFP EC00406
CALL JOB:SEARCH-R1-S13D
SET P042 P006
SFTON3D P042
SMOVL C00407 BC00407 V=166.7  +MOVJ EC00407
MOVL C00408 BC00408 V=1000.0  +MOVJ EC00408 VJ=100.00
'EndPath S4005
'Path S4004
SFTOF3D
MOVJ C00409 BC00409 VJ=100.00  +MOVJ EC00409 VJ=100.00
MOVJ C00410 BC00410 VJ=100.00  +MOVJ EC00410 VJ=100.00
MOVJ C00411 BC00411 VJ=100.00  +MOVJ EC00411 VJ=100.00
MOVJ C00412 BC00412 VJ=100.00  +MOVJ EC00412 VJ=100.00
'Path W4635
SFTOF3D
SFTON3D P051
MOVJ C00413 BC00413 VJ=100.00  +MOVJ EC00413 VJ=100.00
SMOVL C00414 BC00414 V=800.0  +MOVJ EC00414
SMOVL C00415 BC00415 V=150.0 PL=0  +MOVJ EC00415
MACRO1 MJ#(0) ARGF14
ARCON
SMOVL C00416 BC00416 V=11.7  +MOVJ EC00416
ARCOF
SMOVL C00417 BC00417 V=800.0  +MOVJ EC00417
SMOVL C00418 BC00418 V=1000.0  +MOVJ EC00418
MOVJ C00419 BC00419 VJ=100.00  +MOVJ EC00419 VJ=100.00
MOVJ C00420 BC00420 VJ=100.00  +MOVJ EC00420 VJ=100.00
SMOVL C00421 BC00421 V=250.0  +MOVJ EC00421
ARCON
SMOVL C00422 BC00422 V=11.7  +MOVJ EC00422
SMOVL C00423 BC00423 V=11.7  +MOVJ EC00423
ARCOF
SMOVL C00424 BC00424 V=166.7  +MOVJ EC00424
SMOVL C00425 BC00425 V=166.7  +MOVJ EC00425
SMOVL C00426 BC00426 V=166.7  +MOVJ EC00426
ARCON
SMOVL C00427 BC00427 V=9.2  +MOVJ EC00427
ARCOF
SMOVL C00428 BC00428 V=133.3  +MOVJ EC00428
SMOVL C00429 BC00429 V=666.7  +MOVJ EC00429
SFTOF3D
'EndPath W4635
'Path W4636
SFTOF3D
SFTON3D P045
MOVJ C00430 BC00430 VJ=100.00  +MOVJ EC00430 VJ=100.00
SMOVL C00431 BC00431 V=800.0  +MOVJ EC00431
SMOVL C00432 BC00432 V=150.0 PL=0  +MOVJ EC00432
MACRO1 MJ#(0) ARGF21
ARCON
SMOVL C00433 BC00433 V=11.7  +MOVJ EC00433
SMOVL C00434 BC00434 V=11.7  +MOVJ EC00434
ARCOF
SMOVL C00435 BC00435 V=800.0  +MOVJ EC00435
SMOVL C00436 BC00436 V=1000.0  +MOVJ EC00436
SFTOF3D
'EndPath W4636
'Path W4637
SFTOF3D
SFTON3D P045
MOVJ C00437 BC00437 VJ=100.00  +MOVJ EC00437 VJ=100.00
SMOVL C00438 BC00438 V=800.0  +MOVJ EC00438
SMOVL C00439 BC00439 V=150.0 PL=0  +MOVJ EC00439
ARCON
SMOVL C00440 BC00440 V=11.7  +MOVJ EC00440
SMOVL C00441 BC00441 V=11.7  +MOVJ EC00441
ARCOF
SMOVL C00442 BC00442 V=800.0  +MOVJ EC00442
SMOVL C00443 BC00443 V=1000.0  +MOVJ EC00443
SFTOF3D
'EndPath W4637
'Path W4638
SFTOF3D
SFTON3D P049
MOVJ C00444 BC00444 VJ=100.00  +MOVJ EC00444 VJ=100.00
SMOVL C00445 BC00445 V=800.0  +MOVJ EC00445
SMOVL C00446 BC00446 V=150.0 PL=0  +MOVJ EC00446
ARCON
SMOVL C00447 BC00447 V=10.0  +MOVJ EC00447
ARCOF
SMOVL C00448 BC00448 V=800.0  +MOVJ EC00448
SMOVL C00449 BC00449 V=1000.0  +MOVJ EC00449
SFTOF3D
'EndPath W4638
'Path W4639
SFTOF3D
SFTON3D P050
MOVJ C00450 BC00450 VJ=100.00  +MOVJ EC00450 VJ=100.00
SMOVL C00451 BC00451 V=800.0  +MOVJ EC00451
SMOVL C00452 BC00452 V=150.0 PL=0  +MOVJ EC00452
ARCON
SMOVL C00453 BC00453 V=11.7  +MOVJ EC00453
ARCOF
SMOVL C00454 BC00454 V=800.0  +MOVJ EC00454
SMOVL C00455 BC00455 V=1000.0  +MOVJ EC00455
SFTOF3D
'EndPath W4639
MOVJ C00456 BC00456 VJ=100.00  +MOVJ EC00456 VJ=100.00
'Path W4640
SFTOF3D
SFTON3D P048
MOVJ C00457 BC00457 VJ=100.00  +MOVJ EC00457 VJ=100.00
SMOVL C00458 BC00458 V=800.0  +MOVJ EC00458
SMOVL C00459 BC00459 V=150.0 PL=0  +MOVJ EC00459
ARCON
SMOVL C00460 BC00460 V=11.7  +MOVJ EC00460
ARCOF
SMOVL C00461 BC00461 V=800.0  +MOVJ EC00461
SMOVL C00462 BC00462 V=1000.0  +MOVJ EC00462
SFTOF3D
'EndPath W4640
'Path W4641
SFTOF3D
SFTON3D P048
MOVJ C00463 BC00463 VJ=100.00  +MOVJ EC00463 VJ=100.00
SMOVL C00464 BC00464 V=800.0  +MOVJ EC00464
SMOVL C00465 BC00465 V=150.0 PL=0  +MOVJ EC00465
ARCON
SMOVL C00466 BC00466 V=11.7  +MOVJ EC00466
ARCOF
SMOVL C00467 BC00467 V=800.0  +MOVJ EC00467
SMOVL C00468 BC00468 V=1000.0  +MOVJ EC00468
SFTOF3D
'EndPath W4641
'Path W4642
SFTOF3D
SFTON3D P047
MOVJ C00469 BC00469 VJ=100.00  +MOVJ EC00469 VJ=100.00
SMOVL C00470 BC00470 V=800.0  +MOVJ EC00470
SMOVL C00471 BC00471 V=150.0 PL=0  +MOVJ EC00471
ARCON
SMOVL C00472 BC00472 V=11.7  +MOVJ EC00472
ARCOF
SMOVL C00473 BC00473 V=800.0  +MOVJ EC00473
SMOVL C00474 BC00474 V=1000.0  +MOVJ EC00474
SFTOF3D
'EndPath W4642
MOVJ C00475 BC00475 VJ=100.00  +MOVJ EC00475 VJ=100.00
MOVJ C00476 BC00476 VJ=100.00  +MOVJ EC00476 VJ=100.00
'Path W4643
SFTOF3D
SFTON3D P043
MOVJ C00477 BC00477 VJ=100.00  +MOVJ EC00477 VJ=100.00
SMOVL C00478 BC00478 V=800.0  +MOVJ EC00478
SMOVL C00479 BC00479 V=150.0 PL=0  +MOVJ EC00479
ARCON
SMOVL C00480 BC00480 V=11.7  +MOVJ EC00480
ARCOF
SMOVL C00481 BC00481 V=800.0  +MOVJ EC00481
SMOVL C00482 BC00482 V=1000.0  +MOVJ EC00482
SFTOF3D
'EndPath W4643
'Path W4644
SFTOF3D
SFTON3D P043
MOVJ C00483 BC00483 VJ=100.00  +MOVJ EC00483 VJ=100.00
SMOVL C00484 BC00484 V=800.0  +MOVJ EC00484
SMOVL C00485 BC00485 V=150.0 PL=0  +MOVJ EC00485
ARCON
SMOVL C00486 BC00486 V=11.7  +MOVJ EC00486
ARCOF
SMOVL C00487 BC00487 V=800.0  +MOVJ EC00487
SMOVL C00488 BC00488 V=1000.0  +MOVJ EC00488
SFTOF3D
'EndPath W4644
'Path W4645
SFTOF3D
SFTON3D P042
MOVJ C00489 BC00489 VJ=100.00  +MOVJ EC00489 VJ=100.00
SMOVL C00490 BC00490 V=800.0  +MOVJ EC00490
SMOVL C00491 BC00491 V=150.0 PL=0  +MOVJ EC00491
ARCON
SMOVL C00492 BC00492 V=11.7  +MOVJ EC00492
ARCOF
SMOVL C00493 BC00493 V=800.0  +MOVJ EC00493
SMOVL C00494 BC00494 V=1000.0  +MOVJ EC00494
SFTOF3D
'EndPath W4645
'Path W4646
SFTOF3D
SFTON3D P042
MOVJ C00495 BC00495 VJ=100.00  +MOVJ EC00495 VJ=100.00
SMOVL C00496 BC00496 V=800.0  +MOVJ EC00496
SMOVL C00497 BC00497 V=150.0 PL=0  +MOVJ EC00497
ARCON
SMOVL C00498 BC00498 V=11.7  +MOVJ EC00498
ARCOF
SMOVL C00499 BC00499 V=800.0  +MOVJ EC00499
SMOVL C00500 BC00500 V=1000.0  +MOVJ EC00500
SFTOF3D
'EndPath W4646
'3
MOVJ C00501 BC00501 VJ=100.00  +MOVJ EC00501 VJ=100.00
MOVJ C00502 BC00502 VJ=100.00  +MOVJ EC00502 VJ=100.00
'Path W4647
SFTOF3D
SFTON3D P044
MOVJ C00503 BC00503 VJ=100.00  +MOVJ EC00503 VJ=100.00
SMOVL C00504 BC00504 V=800.0  +MOVJ EC00504
SMOVL C00505 BC00505 V=150.0 PL=0  +MOVJ EC00505
ARCON
SMOVL C00506 BC00506 V=11.7  +MOVJ EC00506
ARCOF
SMOVL C00507 BC00507 V=800.0  +MOVJ EC00507
SMOVL C00508 BC00508 V=1000.0  +MOVJ EC00508
SFTOF3D
'EndPath W4647
'Path W4648
SFTOF3D
SFTON3D P046
MOVJ C00509 BC00509 VJ=100.00  +MOVJ EC00509 VJ=100.00
SMOVL C00510 BC00510 V=800.0  +MOVJ EC00510
SMOVL C00511 BC00511 V=150.0 PL=0  +MOVJ EC00511
MACRO1 MJ#(0) ARGF14
ARCON
SMOVL C00512 BC00512 V=11.7  +MOVJ EC00512
ARCOF
SMOVL C00513 BC00513 V=800.0  +MOVJ EC00513
SMOVL C00514 BC00514 V=1000.0  +MOVJ EC00514
SFTOF3D
'EndPath W4648
MOVJ C00515 BC00515 VJ=100.00  +MOVJ EC00515 VJ=100.00
MOVJ C00516 BC00516 VJ=100.00  +MOVJ EC00516 VJ=100.00
END
